;FOLD PLACE 14
;FOLD PROPRIEDADES
MatrizPontos[Pallet_1,Prdt_15CoffeCrisp,14].NumCaixas = 3
MatrizPontos[Pallet_1,Prdt_15CoffeCrisp,14].PickOp = 6
MatrizPontos[Pallet_1,Prdt_15CoffeCrisp,14].ConfGarraOp = 5
MatrizPontos[Pallet_1,Prdt_15CoffeCrisp,14].FechaGarraOp = 0
MatrizPontos[Pallet_1,Prdt_15CoffeCrisp,14].AbreGarraOp = 1
MatrizPontos[Pallet_1,Prdt_15CoffeCrisp,14].SensoresCaixa = 1234
MatrizPontos[Pallet_1,Prdt_15CoffeCrisp,14].TravaGarra = True
MatrizPontos[Pallet_1,Prdt_15CoffeCrisp,14].SkipGoHome = False
MatrizPontos[Pallet_1,Prdt_15CoffeCrisp,14].SkipSobeRelAtual = False
MatrizPontos[Pallet_1,Prdt_15CoffeCrisp,14].XApp1Place=P1_15CoffeCrisp_14_App1
MatrizPontos[Pallet_1,Prdt_15CoffeCrisp,14].XApp2Place=P1_15CoffeCrisp_14_App2
MatrizPontos[Pallet_1,Prdt_15CoffeCrisp,14].XPlace=P1_15CoffeCrisp_14_Place
;ENDFOLD
;FOLD OffsetPlace
MatrizPontos[Pallet_1,Prdt_15CoffeCrisp,14].OffsetPlace.X=0
MatrizPontos[Pallet_1,Prdt_15CoffeCrisp,14].OffsetPlace.Y=0
MatrizPontos[Pallet_1,Prdt_15CoffeCrisp,14].OffsetPlace.Z=0
MatrizPontos[Pallet_1,Prdt_15CoffeCrisp,14].OffsetPlace.A=0
MatrizPontos[Pallet_1,Prdt_15CoffeCrisp,14].OffsetPlace.B=0
MatrizPontos[Pallet_1,Prdt_15CoffeCrisp,14].OffsetPlace.C=0
;ENDFOLD
;ENDFOLD

;ENDFOLD
;ENDFOLD

;FOLD Pallet 1 - Produto 7Aero
;FOLD LAYER 1: PLACE 1 ate 8
;FOLD PLACE 1
;FOLD PROPRIEDADES
MatrizPontos[Pallet_1,Prdt_7Aero,1].NumCaixas = 3
MatrizPontos[Pallet_1,Prdt_7Aero,1].PickOp = 6
MatrizPontos[Pallet_1,Prdt_7Aero,1].ConfGarraOp = 0
MatrizPontos[Pallet_1,Prdt_7Aero,1].FechaGarraOp = 0
MatrizPontos[Pallet_1,Prdt_7Aero,1].AbreGarraOp = 0
MatrizPontos[Pallet_1,Prdt_7Aero,1].SensoresCaixa = 564
MatrizPontos[Pallet_1,Prdt_7Aero,1].TravaGarra = False
MatrizPontos[Pallet_1,Prdt_7Aero,1].SkipGoHome = False
MatrizPontos[Pallet_1,Prdt_7Aero,1].SkipSobeRelAtual = False
MatrizPontos[Pallet_1,Prdt_7Aero,1].XApp1Place=P1_7Aero_1_App1
MatrizPontos[Pallet_1,Prdt_7Aero,1].XApp2Place=P1_7Aero_1_App2
MatrizPontos[Pallet_1,Prdt_7Aero,1].XPlace=P1_7Aero_1_Place
;ENDFOLD
;FOLD OffsetPlace
MatrizPontos[Pallet_1,Prdt_7Aero,1].OffsetPlace.X=0
MatrizPontos[Pallet_1,Prdt_7Aero,1].OffsetPlace.Y=0
MatrizPontos[Pallet_1,Prdt_7Aero,1].OffsetPlace.Z=0
MatrizPontos[Pallet_1,Prdt_7Aero,1].OffsetPlace.A=0
MatrizPontos[Pallet_1,Prdt_7Aero,1].OffsetPlace.B=0
MatrizPontos[Pallet_1,Prdt_7Aero,1].OffsetPlace.C=0
;ENDFOLD
;ENDFOLD

;FOLD PLACE 2
;FOLD PROPRIEDADES
MatrizPontos[Pallet_1,Prdt_7Aero,2].NumCaixas = 3
MatrizPontos[Pallet_1,Prdt_7Aero,2].PickOp = 6
MatrizPontos[Pallet_1,Prdt_7Aero,2].ConfGarraOp = 0
MatrizPontos[Pallet_1,Prdt_7Aero,2].FechaGarraOp = 0
MatrizPontos[Pallet_1,Prdt_7Aero,2].AbreGarraOp = 0
MatrizPontos[Pallet_1,Prdt_7Aero,2].SensoresCaixa = 564
MatrizPontos[Pallet_1,Prdt_7Aero,2].TravaGarra = False
MatrizPontos[Pallet_1,Prdt_7Aero,2].SkipGoHome = False
MatrizPontos[Pallet_1,Prdt_7Aero,2].SkipSobeRelAtual = False
MatrizPontos[Pallet_1,Prdt_7Aero,2].XApp1Place=P1_7Aero_2_App1
MatrizPontos[Pallet_1,Prdt_7Aero,2].XApp2Place=P1_7Aero_2_App2
MatrizPontos[Pallet_1,Prdt_7Aero,2].XPlace=P1_7Aero_2_Place
;ENDFOLD
;FOLD OffsetPlace
MatrizPontos[Pallet_1,Prdt_7Aero,2].OffsetPlace.X=0
MatrizPontos[Pallet_1,Prdt_7Aero,2].OffsetPlace.Y=0
MatrizPontos[Pallet_1,Prdt_7Aero,2].OffsetPlace.Z=0
MatrizPontos[Pallet_1,Prdt_7Aero,2].OffsetPlace.A=0
MatrizPontos[Pallet_1,Prdt_7Aero,2].OffsetPlace.B=0
MatrizPontos[Pallet_1,Prdt_7Aero,2].OffsetPlace.C=0
;ENDFOLD
;ENDFOLD

;FOLD PLACE 3
;FOLD PROPRIEDADES
MatrizPontos[Pallet_1,Prdt_7Aero,3].NumCaixas = 2
MatrizPontos[Pallet_1,Prdt_7Aero,3].PickOp = 8
MatrizPontos[Pallet_1,Prdt_7Aero,3].ConfGarraOp = 5
MatrizPontos[Pallet_1,Prdt_7Aero,3].FechaGarraOp = 0
MatrizPontos[Pallet_1,Prdt_7Aero,3].AbreGarraOp = 0
MatrizPontos[Pallet_1,Prdt_7Aero,3].SensoresCaixa = 12
MatrizPontos[Pallet_1,Prdt_7Aero,3].TravaGarra = False
MatrizPontos[Pallet_1,Prdt_7Aero,3].SkipGoHome = False
MatrizPontos[Pallet_1,Prdt_7Aero,3].SkipSobeRelAtual = False
MatrizPontos[Pallet_1,Prdt_7Aero,3].XApp1Place=P1_7Aero_3_App1
MatrizPontos[Pallet_1,Prdt_7Aero,3].XApp2Place=P1_7Aero_3_App2
MatrizPontos[Pallet_1,Prdt_7Aero,3].XPlace=P1_7Aero_3_Place
;ENDFOLD
;FOLD OffsetPlace
MatrizPontos[Pallet_1,Prdt_7Aero,3].OffsetPlace.X=0
MatrizPontos[Pallet_1,Prdt_7Aero,3].OffsetPlace.Y=0
MatrizPontos[Pallet_1,Prdt_7Aero,3].OffsetPlace.Z=0
MatrizPontos[Pallet_1,Prdt_7Aero,3].OffsetPlace.A=0
MatrizPontos[Pallet_1,Prdt_7Aero,3].OffsetPlace.B=0
MatrizPontos[Pallet_1,Prdt_7Aero,3].OffsetPlace.C=0
;ENDFOLD
;ENDFOLD

;FOLD PLACE 4
;FOLD PROPRIEDADES
MatrizPontos[Pallet_1,Prdt_7Aero,4].NumCaixas = 2
MatrizPontos[Pallet_1,Prdt_7Aero,4].PickOp = 8
MatrizPontos[Pallet_1,Prdt_7Aero,4].ConfGarraOp = 5
MatrizPontos[Pallet_1,Prdt_7Aero,4].FechaGarraOp = 0
MatrizPontos[Pallet_1,Prdt_7Aero,4].AbreGarraOp = 0
MatrizPontos[Pallet_1,Prdt_7Aero,4].SensoresCaixa = 12
MatrizPontos[Pallet_1,Prdt_7Aero,4].TravaGarra = False
MatrizPontos[Pallet_1,Prdt_7Aero,4].SkipGoHome = False
MatrizPontos[Pallet_1,Prdt_7Aero,4].SkipSobeRelAtual = False
MatrizPontos[Pallet_1,Prdt_7Aero,4].XApp1Place=P1_7Aero_4_App1
MatrizPontos[Pallet_1,Prdt_7Aero,4].XApp2Place=P1_7Aero_4_App2
MatrizPontos[Pallet_1,Prdt_7Aero,4].XPlace=P1_7Aero_4_Place
;ENDFOLD
;FOLD OffsetPlace
MatrizPontos[Pallet_1,Prdt_7Aero,4].OffsetPlace.X=0
MatrizPontos[Pallet_1,Prdt_7Aero,4].OffsetPlace.Y=0
MatrizPontos[Pallet_1,Prdt_7Aero,4].OffsetPlace.Z=0
MatrizPontos[Pallet_1,Prdt_7Aero,4].OffsetPlace.A=0
MatrizPontos[Pallet_1,Prdt_7Aero,4].OffsetPlace.B=0
MatrizPontos[Pallet_1,Prdt_7Aero,4].OffsetPlace.C=0
;ENDFOLD
;ENDFOLD

;FOLD PLACE 5
;FOLD PROPRIEDADES
MatrizPontos[Pallet_1,Prdt_7Aero,5].NumCaixas = 3
MatrizPontos[Pallet_1,Prdt_7Aero,5].PickOp = 8
MatrizPontos[Pallet_1,Prdt_7Aero,5].ConfGarraOp = 5
MatrizPontos[Pallet_1,Prdt_7Aero,5].FechaGarraOp = 0
MatrizPontos[Pallet_1,Prdt_7Aero,5].AbreGarraOp = 1
MatrizPontos[Pallet_1,Prdt_7Aero,5].SensoresCaixa = 123
MatrizPontos[Pallet_1,Prdt_7Aero,5].TravaGarra = True
MatrizPontos[Pallet_1,Prdt_7Aero,5].SkipGoHome = False
MatrizPontos[Pallet_1,Prdt_7Aero,5].SkipSobeRelAtual = False
MatrizPontos[Pallet_1,Prdt_7Aero,5].XApp1Place=P1_7Aero_5_App1
MatrizPontos[Pallet_1,Prdt_7Aero,5].XApp2Place=P1_7Aero_5_App2
MatrizPontos[Pallet_1,Prdt_7Aero,5].XPlace=P1_7Aero_5_Place
;ENDFOLD
;FOLD OffsetPlace
MatrizPontos[Pallet_1,Prdt_7Aero,5].OffsetPlace.X=0
MatrizPontos[Pallet_1,Prdt_7Aero,5].OffsetPlace.Y=0
MatrizPontos[Pallet_1,Prdt_7Aero,5].OffsetPlace.Z=0
MatrizPontos[Pallet_1,Prdt_7Aero,5].OffsetPlace.A=0
MatrizPontos[Pallet_1,Prdt_7Aero,5].OffsetPlace.B=0
MatrizPontos[Pallet_1,Prdt_7Aero,5].OffsetPlace.C=0
;ENDFOLD
;ENDFOLD

;FOLD PLACE 6
;FOLD PROPRIEDADES
MatrizPontos[Pallet_1,Prdt_7Aero,6].NumCaixas = 3
MatrizPontos[Pallet_1,Prdt_7Aero,6].PickOp = 8
MatrizPontos[Pallet_1,Prdt_7Aero,6].ConfGarraOp = 5
MatrizPontos[Pallet_1,Prdt_7Aero,6].FechaGarraOp = 0
MatrizPontos[Pallet_1,Prdt_7Aero,6].AbreGarraOp = 1
MatrizPontos[Pallet_1,Prdt_7Aero,6].SensoresCaixa = 123
MatrizPontos[Pallet_1,Prdt_7Aero,6].TravaGarra = True
MatrizPontos[Pallet_1,Prdt_7Aero,6].SkipGoHome = False
MatrizPontos[Pallet_1,Prdt_7Aero,6].SkipSobeRelAtual = False
MatrizPontos[Pallet_1,Prdt_7Aero,6].XApp1Place=P1_7Aero_6_App1
MatrizPontos[Pallet_1,Prdt_7Aero,6].XApp2Place=P1_7Aero_6_App2
MatrizPontos[Pallet_1,Prdt_7Aero,6].XPlace=P1_7Aero_6_Place
;ENDFOLD
;FOLD OffsetPlace
MatrizPontos[Pallet_1,Prdt_7Aero,6].OffsetPlace.X=0
MatrizPontos[Pallet_1,Prdt_7Aero,6].OffsetPlace.Y=0
MatrizPontos[Pallet_1,Prdt_7Aero,6].OffsetPlace.Z=0
MatrizPontos[Pallet_1,Prdt_7Aero,6].OffsetPlace.A=0
MatrizPontos[Pallet_1,Prdt_7Aero,6].OffsetPlace.B=0
MatrizPontos[Pallet_1,Prdt_7Aero,6].OffsetPlace.C=0
;ENDFOLD
;ENDFOLD

;FOLD PLACE 7
;FOLD PROPRIEDADES
MatrizPontos[Pallet_1,Prdt_7Aero,7].NumCaixas = 2
MatrizPontos[Pallet_1,Prdt_7Aero,7].PickOp = 8
MatrizPontos[Pallet_1,Prdt_7Aero,7].ConfGarraOp = 5
MatrizPontos[Pallet_1,Prdt_7Aero,7].FechaGarraOp = 0
MatrizPontos[Pallet_1,Prdt_7Aero,7].AbreGarraOp = 1
MatrizPontos[Pallet_1,Prdt_7Aero,7].SensoresCaixa = 12
MatrizPontos[Pallet_1,Prdt_7Aero,7].TravaGarra = True
MatrizPontos[Pallet_1,Prdt_7Aero,7].SkipGoHome = False
MatrizPontos[Pallet_1,Prdt_7Aero,7].SkipSobeRelAtual = False
MatrizPontos[Pallet_1,Prdt_7Aero,7].XApp1Place=P1_7Aero_7_App1
MatrizPontos[Pallet_1,Prdt_7Aero,7].XApp2Place=P1_7Aero_7_App2
MatrizPontos[Pallet_1,Prdt_7Aero,7].XPlace=P1_7Aero_7_Place
;ENDFOLD
;FOLD OffsetPlace
MatrizPontos[Pallet_1,Prdt_7Aero,7].OffsetPlace.X=0
MatrizPontos[Pallet_1,Prdt_7Aero,7].OffsetPlace.Y=0
MatrizPontos[Pallet_1,Prdt_7Aero,7].OffsetPlace.Z=0
MatrizPontos[Pallet_1,Prdt_7Aero,7].OffsetPlace.A=0
MatrizPontos[Pallet_1,Prdt_7Aero,7].OffsetPlace.B=0
MatrizPontos[Pallet_1,Prdt_7Aero,7].OffsetPlace.C=0
;ENDFOLD
;ENDFOLD

;FOLD PLACE 8
;FOLD PROPRIEDADES
MatrizPontos[Pallet_1,Prdt_7Aero,8].NumCaixas = 2
MatrizPontos[Pallet_1,Prdt_7Aero,8].PickOp = 8
MatrizPontos[Pallet_1,Prdt_7Aero,8].ConfGarraOp = 5
MatrizPontos[Pallet_1,Prdt_7Aero,8].FechaGarraOp = 0
MatrizPontos[Pallet_1,Prdt_7Aero,8].AbreGarraOp = 1
MatrizPontos[Pallet_1,Prdt_7Aero,8].SensoresCaixa = 12
MatrizPontos[Pallet_1,Prdt_7Aero,8].TravaGarra = True
MatrizPontos[Pallet_1,Prdt_7Aero,8].SkipGoHome = False
MatrizPontos[Pallet_1,Prdt_7Aero,8].SkipSobeRelAtual = False
MatrizPontos[Pallet_1,Prdt_7Aero,8].XApp1Place=P1_7Aero_8_App1
MatrizPontos[Pallet_1,Prdt_7Aero,8].XApp2Place=P1_7Aero_8_App2
MatrizPontos[Pallet_1,Prdt_7Aero,8].XPlace=P1_7Aero_8_Place
;ENDFOLD
;FOLD OffsetPlace
MatrizPontos[Pallet_1,Prdt_7Aero,8].OffsetPlace.X=0
MatrizPontos[Pallet_1,Prdt_7Aero,8].OffsetPlace.Y=0
MatrizPontos[Pallet_1,Prdt_7Aero,8].OffsetPlace.Z=0
MatrizPontos[Pallet_1,Prdt_7Aero,8].OffsetPlace.A=0
MatrizPontos[Pallet_1,Prdt_7Aero,8].OffsetPlace.B=0
MatrizPontos[Pallet_1,Prdt_7Aero,8].OffsetPlace.C=0
;ENDFOLD
;ENDFOLD

;ENDFOLD
;FOLD LAYER 2: PLACE 9 ate 16
;FOLD PLACE 9
;FOLD PROPRIEDADES
MatrizPontos[Pallet_1,Prdt_7Aero,9].NumCaixas = 2
MatrizPontos[Pallet_1,Prdt_7Aero,9].PickOp = 8
MatrizPontos[Pallet_1,Prdt_7Aero,9].ConfGarraOp = 5
MatrizPontos[Pallet_1,Prdt_7Aero,9].FechaGarraOp = 0
MatrizPontos[Pallet_1,Prdt_7Aero,9].AbreGarraOp = 1
MatrizPontos[Pallet_1,Prdt_7Aero,9].SensoresCaixa = 12
MatrizPontos[Pallet_1,Prdt_7Aero,9].TravaGarra = True
MatrizPontos[Pallet_1,Prdt_7Aero,9].SkipGoHome = False
MatrizPontos[Pallet_1,Prdt_7Aero,9].SkipSobeRelAtual = False
MatrizPontos[Pallet_1,Prdt_7Aero,9].XApp1Place=P1_7Aero_9_App1
MatrizPontos[Pallet_1,Prdt_7Aero,9].XApp2Place=P1_7Aero_9_App2
MatrizPontos[Pallet_1,Prdt_7Aero,9].XPlace=P1_7Aero_9_Place
;ENDFOLD
;FOLD OffsetPlace
MatrizPontos[Pallet_1,Prdt_7Aero,9].OffsetPlace.X=0
MatrizPontos[Pallet_1,Prdt_7Aero,9].OffsetPlace.Y=0
MatrizPontos[Pallet_1,Prdt_7Aero,9].OffsetPlace.Z=0
MatrizPontos[Pallet_1,Prdt_7Aero,9].OffsetPlace.A=0
MatrizPontos[Pallet_1,Prdt_7Aero,9].OffsetPlace.B=0
MatrizPontos[Pallet_1,Prdt_7Aero,9].OffsetPlace.C=0
;ENDFOLD
;ENDFOLD

;FOLD PLACE 10
;FOLD PROPRIEDADES
MatrizPontos[Pallet_1,Prdt_7Aero,10].NumCaixas = 2
MatrizPontos[Pallet_1,Prdt_7Aero,10].PickOp = 8
MatrizPontos[Pallet_1,Prdt_7Aero,10].ConfGarraOp = 5
MatrizPontos[Pallet_1,Prdt_7Aero,10].FechaGarraOp = 0
MatrizPontos[Pallet_1,Prdt_7Aero,10].AbreGarraOp = 1
MatrizPontos[Pallet_1,Prdt_7Aero,10].SensoresCaixa = 12
MatrizPontos[Pallet_1,Prdt_7Aero,10].TravaGarra = True
MatrizPontos[Pallet_1,Prdt_7Aero,10].SkipGoHome = False
MatrizPontos[Pallet_1,Prdt_7Aero,10].SkipSobeRelAtual = False
MatrizPontos[Pallet_1,Prdt_7Aero,10].XApp1Place=P1_7Aero_10_App1
MatrizPontos[Pallet_1,Prdt_7Aero,10].XApp2Place=P1_7Aero_10_App2
MatrizPontos[Pallet_1,Prdt_7Aero,10].XPlace=P1_7Aero_10_Place
;ENDFOLD
;FOLD OffsetPlace
MatrizPontos[Pallet_1,Prdt_7Aero,10].OffsetPlace.X=0
MatrizPontos[Pallet_1,Prdt_7Aero,10].OffsetPlace.Y=0
MatrizPontos[Pallet_1,Prdt_7Aero,10].OffsetPlace.Z=0
MatrizPontos[Pallet_1,Prdt_7Aero,10].OffsetPlace.A=0
MatrizPontos[Pallet_1,Prdt_7Aero,10].OffsetPlace.B=0
MatrizPontos[Pallet_1,Prdt_7Aero,10].OffsetPlace.C=0
;ENDFOLD
;ENDFOLD

;FOLD PLACE 11
;FOLD PROPRIEDADES
MatrizPontos[Pallet_1,Prdt_7Aero,11].NumCaixas = 3
MatrizPontos[Pallet_1,Prdt_7Aero,11].PickOp = 8
MatrizPontos[Pallet_1,Prdt_7Aero,11].ConfGarraOp = 5
MatrizPontos[Pallet_1,Prdt_7Aero,11].FechaGarraOp = 0
MatrizPontos[Pallet_1,Prdt_7Aero,11].AbreGarraOp = 0
MatrizPontos[Pallet_1,Prdt_7Aero,11].SensoresCaixa = 123
MatrizPontos[Pallet_1,Prdt_7Aero,11].TravaGarra = False
MatrizPontos[Pallet_1,Prdt_7Aero,11].SkipGoHome = False
MatrizPontos[Pallet_1,Prdt_7Aero,11].SkipSobeRelAtual = False
MatrizPontos[Pallet_1,Prdt_7Aero,11].XApp1Place=P1_7Aero_11_App1
MatrizPontos[Pallet_1,Prdt_7Aero,11].XApp2Place=P1_7Aero_11_App2
MatrizPontos[Pallet_1,Prdt_7Aero,11].XPlace=P1_7Aero_11_Place
;ENDFOLD
;FOLD OffsetPlace
MatrizPontos[Pallet_1,Prdt_7Aero,11].OffsetPlace.X=0
MatrizPontos[Pallet_1,Prdt_7Aero,11].OffsetPlace.Y=0
MatrizPontos[Pallet_1,Prdt_7Aero,11].OffsetPlace.Z=0
MatrizPontos[Pallet_1,Prdt_7Aero,11].OffsetPlace.A=0
MatrizPontos[Pallet_1,Prdt_7Aero,11].OffsetPlace.B=0
MatrizPontos[Pallet_1,Prdt_7Aero,11].OffsetPlace.C=0
;ENDFOLD
;ENDFOLD

;FOLD PLACE 12
;FOLD PROPRIEDADES
MatrizPontos[Pallet_1,Prdt_7Aero,12].NumCaixas = 3
MatrizPontos[Pallet_1,Prdt_7Aero,12].PickOp = 8
MatrizPontos[Pallet_1,Prdt_7Aero,12].ConfGarraOp = 5
MatrizPontos[Pallet_1,Prdt_7Aero,12].FechaGarraOp = 0
MatrizPontos[Pallet_1,Prdt_7Aero,12].AbreGarraOp = 0
MatrizPontos[Pallet_1,Prdt_7Aero,12].SensoresCaixa = 123
MatrizPontos[Pallet_1,Prdt_7Aero,12].TravaGarra = False
MatrizPontos[Pallet_1,Prdt_7Aero,12].SkipGoHome = False
MatrizPontos[Pallet_1,Prdt_7Aero,12].SkipSobeRelAtual = False
MatrizPontos[Pallet_1,Prdt_7Aero,12].XApp1Place=P1_7Aero_12_App1
MatrizPontos[Pallet_1,Prdt_7Aero,12].XApp2Place=P1_7Aero_12_App2
MatrizPontos[Pallet_1,Prdt_7Aero,12].XPlace=P1_7Aero_12_Place
;ENDFOLD
;FOLD OffsetPlace
MatrizPontos[Pallet_1,Prdt_7Aero,12].OffsetPlace.X=0
MatrizPontos[Pallet_1,Prdt_7Aero,12].OffsetPlace.Y=0
MatrizPontos[Pallet_1,Prdt_7Aero,12].OffsetPlace.Z=0
MatrizPontos[Pallet_1,Prdt_7Aero,12].OffsetPlace.A=0
MatrizPontos[Pallet_1,Prdt_7Aero,12].OffsetPlace.B=0
MatrizPontos[Pallet_1,Prdt_7Aero,12].OffsetPlace.C=0
;ENDFOLD
;ENDFOLD

;FOLD PLACE 13
;FOLD PROPRIEDADES
MatrizPontos[Pallet_1,Prdt_7Aero,13].NumCaixas = 3
MatrizPontos[Pallet_1,Prdt_7Aero,13].PickOp = 8
MatrizPontos[Pallet_1,Prdt_7Aero,13].ConfGarraOp = 5
MatrizPontos[Pallet_1,Prdt_7Aero,13].FechaGarraOp = 0
MatrizPontos[Pallet_1,Prdt_7Aero,13].AbreGarraOp = 0
MatrizPontos[Pallet_1,Prdt_7Aero,13].SensoresCaixa = 123
MatrizPontos[Pallet_1,Prdt_7Aero,13].TravaGarra = False
MatrizPontos[Pallet_1,Prdt_7Aero,13].SkipGoHome = False
MatrizPontos[Pallet_1,Prdt_7Aero,13].SkipSobeRelAtual = False
MatrizPontos[Pallet_1,Prdt_7Aero,13].XApp1Place=P1_7Aero_13_App1
MatrizPontos[Pallet_1,Prdt_7Aero,13].XApp2Place=P1_7Aero_13_App2
MatrizPontos[Pallet_1,Prdt_7Aero,13].XPlace=P1_7Aero_13_Place
;ENDFOLD
;FOLD OffsetPlace
MatrizPontos[Pallet_1,Prdt_7Aero,13].OffsetPlace.X=0
MatrizPontos[Pallet_1,Prdt_7Aero,13].OffsetPlace.Y=0
MatrizPontos[Pallet_1,Prdt_7Aero,13].OffsetPlace.Z=0
MatrizPontos[Pallet_1,Prdt_7Aero,13].OffsetPlace.A=0
MatrizPontos[Pallet_1,Prdt_7Aero,13].OffsetPlace.B=0
MatrizPontos[Pallet_1,Prdt_7Aero,13].OffsetPlace.C=0
;ENDFOLD
;ENDFOLD

;FOLD PLACE 14
;FOLD PROPRIEDADES
MatrizPontos[Pallet_1,Prdt_7Aero,14].NumCaixas = 3
MatrizPontos[Pallet_1,Prdt_7Aero,14].PickOp = 8
MatrizPontos[Pallet_1,Prdt_7Aero,14].ConfGarraOp = 5
MatrizPontos[Pallet_1,Prdt_7Aero,14].FechaGarraOp = 0
MatrizPontos[Pallet_1,Prdt_7Aero,14].AbreGarraOp = 0
MatrizPontos[Pallet_1,Prdt_7Aero,14].SensoresCaixa = 123
MatrizPontos[Pallet_1,Prdt_7Aero,14].TravaGarra = False
MatrizPontos[Pallet_1,Prdt_7Aero,14].SkipGoHome = False
MatrizPontos[Pallet_1,Prdt_7Aero,14].SkipSobeRelAtual = False
MatrizPontos[Pallet_1,Prdt_7Aero,14].XApp1Place=P1_7Aero_14_App1
MatrizPontos[Pallet_1,Prdt_7Aero,14].XApp2Place=P1_7Aero_14_App2
MatrizPontos[Pallet_1,Prdt_7Aero,14].XPlace=P1_7Aero_14_Place
;ENDFOLD
;FOLD OffsetPlace
MatrizPontos[Pallet_1,Prdt_7Aero,14].OffsetPlace.X=0
MatrizPontos[Pallet_1,Prdt_7Aero,14].OffsetPlace.Y=0
MatrizPontos[Pallet_1,Prdt_7Aero,14].OffsetPlace.Z=0
MatrizPontos[Pallet_1,Prdt_7Aero,14].OffsetPlace.A=0
MatrizPontos[Pallet_1,Prdt_7Aero,14].OffsetPlace.B=0
MatrizPontos[Pallet_1,Prdt_7Aero,14].OffsetPlace.C=0
;ENDFOLD
;ENDFOLD

;FOLD PLACE 15
;FOLD PROPRIEDADES
MatrizPontos[Pallet_1,Prdt_7Aero,15].NumCaixas = 2
MatrizPontos[Pallet_1,Prdt_7Aero,15].PickOp = 8
MatrizPontos[Pallet_1,Prdt_7Aero,15].ConfGarraOp = 5
MatrizPontos[Pallet_1,Prdt_7Aero,15].FechaGarraOp = 0
MatrizPontos[Pallet_1,Prdt_7Aero,15].AbreGarraOp = 1
MatrizPontos[Pallet_1,Prdt_7Aero,15].SensoresCaixa = 12
MatrizPontos[Pallet_1,Prdt_7Aero,15].TravaGarra = True
MatrizPontos[Pallet_1,Prdt_7Aero,15].SkipGoHome = False
MatrizPontos[Pallet_1,Prdt_7Aero,15].SkipSobeRelAtual = False
MatrizPontos[Pallet_1,Prdt_7Aero,15].XApp1Place=P1_7Aero_15_App1
MatrizPontos[Pallet_1,Prdt_7Aero,15].XApp2Place=P1_7Aero_15_App2
MatrizPontos[Pallet_1,Prdt_7Aero,15].XPlace=P1_7Aero_15_Place
;ENDFOLD
;FOLD OffsetPlace
MatrizPontos[Pallet_1,Prdt_7Aero,15].OffsetPlace.X=0
MatrizPontos[Pallet_1,Prdt_7Aero,15].OffsetPlace.Y=0
MatrizPontos[Pallet_1,Prdt_7Aero,15].OffsetPlace.Z=0
MatrizPontos[Pallet_1,Prdt_7Aero,15].OffsetPlace.A=0
MatrizPontos[Pallet_1,Prdt_7Aero,15].OffsetPlace.B=0
MatrizPontos[Pallet_1,Prdt_7Aero,15].OffsetPlace.C=0
;ENDFOLD
;ENDFOLD

;FOLD PLACE 16
;FOLD PROPRIEDADES
MatrizPontos[Pallet_1,Prdt_7Aero,16].NumCaixas = 2
MatrizPontos[Pallet_1,Prdt_7Aero,16].PickOp = 8
MatrizPontos[Pallet_1,Prdt_7Aero,16].ConfGarraOp = 5
MatrizPontos[Pallet_1,Prdt_7Aero,16].FechaGarraOp = 0
MatrizPontos[Pallet_1,Prdt_7Aero,16].AbreGarraOp = 1
MatrizPontos[Pallet_1,Prdt_7Aero,16].SensoresCaixa = 12
MatrizPontos[Pallet_1,Prdt_7Aero,16].TravaGarra = True
MatrizPontos[Pallet_1,Prdt_7Aero,16].SkipGoHome = False
MatrizPontos[Pallet_1,Prdt_7Aero,16].SkipSobeRelAtual = False
MatrizPontos[Pallet_1,Prdt_7Aero,16].XApp1Place=P1_7Aero_16_App1
MatrizPontos[Pallet_1,Prdt_7Aero,16].XApp2Place=P1_7Aero_16_App2
MatrizPontos[Pallet_1,Prdt_7Aero,16].XPlace=P1_7Aero_16_Place
;ENDFOLD
;FOLD OffsetPlace
MatrizPontos[Pallet_1,Prdt_7Aero,16].OffsetPlace.X=0
MatrizPontos[Pallet_1,Prdt_7Aero,16].OffsetPlace.Y=0
MatrizPontos[Pallet_1,Prdt_7Aero,16].OffsetPlace.Z=0
MatrizPontos[Pallet_1,Prdt_7Aero,16].OffsetPlace.A=0
MatrizPontos[Pallet_1,Prdt_7Aero,16].OffsetPlace.B=0
MatrizPontos[Pallet_1,Prdt_7Aero,16].OffsetPlace.C=0
;ENDFOLD
;ENDFOLD

;ENDFOLD
;ENDFOLD

;FOLD Pallet 1 - Produto 32BarPacking
;FOLD LAYER 1: PLACE 1 ate 3
;FOLD PLACE 1
;FOLD PROPRIEDADES
MatrizPontos[Pallet_1,Prdt_32BarPacking,1].NumCaixas = 3
MatrizPontos[Pallet_1,Prdt_32BarPacking,1].PickOp = 2
MatrizPontos[Pallet_1,Prdt_32BarPacking,1].ConfGarraOp = 3
MatrizPontos[Pallet_1,Prdt_32BarPacking,1].FechaGarraOp = 0
MatrizPontos[Pallet_1,Prdt_32BarPacking,1].AbreGarraOp = 0
MatrizPontos[Pallet_1,Prdt_32BarPacking,1].SensoresCaixa = 12345
MatrizPontos[Pallet_1,Prdt_32BarPacking,1].TravaGarra = False
MatrizPontos[Pallet_1,Prdt_32BarPacking,1].SkipGoHome = False
MatrizPontos[Pallet_1,Prdt_32BarPacking,1].SkipSobeRelAtual = False
MatrizPontos[Pallet_1,Prdt_32BarPacking,1].XApp1Place=P1_32BarPacking_1_App1
MatrizPontos[Pallet_1,Prdt_32BarPacking,1].XApp2Place=P1_32BarPacking_1_App2
MatrizPontos[Pallet_1,Prdt_32BarPacking,1].XPlace=P1_32BarPacking_1_Place
;ENDFOLD
;FOLD OffsetPlace
MatrizPontos[Pallet_1,Prdt_32BarPacking,1].OffsetPlace.X=0
MatrizPontos[Pallet_1,Prdt_32BarPacking,1].OffsetPlace.Y=0
MatrizPontos[Pallet_1,Prdt_32BarPacking,1].OffsetPlace.Z=0
MatrizPontos[Pallet_1,Prdt_32BarPacking,1].OffsetPlace.A=0
MatrizPontos[Pallet_1,Prdt_32BarPacking,1].OffsetPlace.B=0
MatrizPontos[Pallet_1,Prdt_32BarPacking,1].OffsetPlace.C=0
;ENDFOLD
;ENDFOLD

;FOLD PLACE 2
;FOLD PROPRIEDADES
MatrizPontos[Pallet_1,Prdt_32BarPacking,2].NumCaixas = 3
MatrizPontos[Pallet_1,Prdt_32BarPacking,2].PickOp = 2
MatrizPontos[Pallet_1,Prdt_32BarPacking,2].ConfGarraOp = 3
MatrizPontos[Pallet_1,Prdt_32BarPacking,2].FechaGarraOp = 0
MatrizPontos[Pallet_1,Prdt_32BarPacking,2].AbreGarraOp = 0
MatrizPontos[Pallet_1,Prdt_32BarPacking,2].SensoresCaixa = 12345
MatrizPontos[Pallet_1,Prdt_32BarPacking,2].TravaGarra = False
MatrizPontos[Pallet_1,Prdt_32BarPacking,2].SkipGoHome = False
MatrizPontos[Pallet_1,Prdt_32BarPacking,2].SkipSobeRelAtual = False
MatrizPontos[Pallet_1,Prdt_32BarPacking,2].XApp1Place=P1_32BarPacking_2_App1
MatrizPontos[Pallet_1,Prdt_32BarPacking,2].XApp2Place=P1_32BarPacking_2_App2
MatrizPontos[Pallet_1,Prdt_32BarPacking,2].XPlace=P1_32BarPacking_2_Place
;ENDFOLD
;FOLD OffsetPlace
MatrizPontos[Pallet_1,Prdt_32BarPacking,2].OffsetPlace.X=0
MatrizPontos[Pallet_1,Prdt_32BarPacking,2].OffsetPlace.Y=0
MatrizPontos[Pallet_1,Prdt_32BarPacking,2].OffsetPlace.Z=0
MatrizPontos[Pallet_1,Prdt_32BarPacking,2].OffsetPlace.A=0
MatrizPontos[Pallet_1,Prdt_32BarPacking,2].OffsetPlace.B=0
MatrizPontos[Pallet_1,Prdt_32BarPacking,2].OffsetPlace.C=0
;ENDFOLD
;ENDFOLD

;FOLD PLACE 3
;FOLD PROPRIEDADES
MatrizPontos[Pallet_1,Prdt_32BarPacking,3].NumCaixas = 3
MatrizPontos[Pallet_1,Prdt_32BarPacking,3].PickOp = 2
MatrizPontos[Pallet_1,Prdt_32BarPacking,3].ConfGarraOp = 3
MatrizPontos[Pallet_1,Prdt_32BarPacking,3].FechaGarraOp = 0
MatrizPontos[Pallet_1,Prdt_32BarPacking,3].AbreGarraOp = 0
MatrizPontos[Pallet_1,Prdt_32BarPacking,3].SensoresCaixa = 12345
MatrizPontos[Pallet_1,Prdt_32BarPacking,3].TravaGarra = False
MatrizPontos[Pallet_1,Prdt_32BarPacking,3].SkipGoHome = False
MatrizPontos[Pallet_1,Prdt_32BarPacking,3].SkipSobeRelAtual = False
MatrizPontos[Pallet_1,Prdt_32BarPacking,3].XApp1Place=P1_32BarPacking_3_App1
MatrizPontos[Pallet_1,Prdt_32BarPacking,3].XApp2Place=P1_32BarPacking_3_App2
MatrizPontos[Pallet_1,Prdt_32BarPacking,3].XPlace=P1_32BarPacking_3_Place
;ENDFOLD
;FOLD OffsetPlace
MatrizPontos[Pallet_1,Prdt_32BarPacking,3].OffsetPlace.X=0
MatrizPontos[Pallet_1,Prdt_32BarPacking,3].OffsetPlace.Y=0
MatrizPontos[Pallet_1,Prdt_32BarPacking,3].OffsetPlace.Z=0
MatrizPontos[Pallet_1,Prdt_32BarPacking,3].OffsetPlace.A=0
MatrizPontos[Pallet_1,Prdt_32BarPacking,3].OffsetPlace.B=0
MatrizPontos[Pallet_1,Prdt_32BarPacking,3].OffsetPlace.C=0
;ENDFOLD
;ENDFOLD

;ENDFOLD
;ENDFOLD

;FOLD Pallet 1 - Produto 33BarPacking
;FOLD LAYER 1: PLACE 1 ate 2
;FOLD PLACE 1
;FOLD PROPRIEDADES
MatrizPontos[Pallet_1,Prdt_33BarPacking,1].NumCaixas = 3
MatrizPontos[Pallet_1,Prdt_33BarPacking,1].PickOp = 2
MatrizPontos[Pallet_1,Prdt_33BarPacking,1].ConfGarraOp = 2
MatrizPontos[Pallet_1,Prdt_33BarPacking,1].FechaGarraOp = 0
MatrizPontos[Pallet_1,Prdt_33BarPacking,1].AbreGarraOp = 0
MatrizPontos[Pallet_1,Prdt_33BarPacking,1].SensoresCaixa = 12345
MatrizPontos[Pallet_1,Prdt_33BarPacking,1].TravaGarra = False
MatrizPontos[Pallet_1,Prdt_33BarPacking,1].SkipGoHome = False
MatrizPontos[Pallet_1,Prdt_33BarPacking,1].SkipSobeRelAtual = False
MatrizPontos[Pallet_1,Prdt_33BarPacking,1].XApp1Place=P1_33BarPacking_1_App1
MatrizPontos[Pallet_1,Prdt_33BarPacking,1].XApp2Place=P1_33BarPacking_1_App2
MatrizPontos[Pallet_1,Prdt_33BarPacking,1].XPlace=P1_33BarPacking_1_Place
;ENDFOLD
;FOLD OffsetPlace
MatrizPontos[Pallet_1,Prdt_33BarPacking,1].OffsetPlace.X=0
MatrizPontos[Pallet_1,Prdt_33BarPacking,1].OffsetPlace.Y=0
MatrizPontos[Pallet_1,Prdt_33BarPacking,1].OffsetPlace.Z=0
MatrizPontos[Pallet_1,Prdt_33BarPacking,1].OffsetPlace.A=0
MatrizPontos[Pallet_1,Prdt_33BarPacking,1].OffsetPlace.B=0
MatrizPontos[Pallet_1,Prdt_33BarPacking,1].OffsetPlace.C=0
;ENDFOLD
;ENDFOLD

;FOLD PLACE 2
;FOLD PROPRIEDADES
MatrizPontos[Pallet_1,Prdt_33BarPacking,2].NumCaixas = 3
MatrizPontos[Pallet_1,Prdt_33BarPacking,2].PickOp = 2
MatrizPontos[Pallet_1,Prdt_33BarPacking,2].ConfGarraOp = 2
MatrizPontos[Pallet_1,Prdt_33BarPacking,2].FechaGarraOp = 0
MatrizPontos[Pallet_1,Prdt_33BarPacking,2].AbreGarraOp = 0
MatrizPontos[Pallet_1,Prdt_33BarPacking,2].SensoresCaixa = 12345
MatrizPontos[Pallet_1,Prdt_33BarPacking,2].TravaGarra = False
MatrizPontos[Pallet_1,Prdt_33BarPacking,2].SkipGoHome = False
MatrizPontos[Pallet_1,Prdt_33BarPacking,2].SkipSobeRelAtual = False
MatrizPontos[Pallet_1,Prdt_33BarPacking,2].XApp1Place=P1_33BarPacking_2_App1
MatrizPontos[Pallet_1,Prdt_33BarPacking,2].XApp2Place=P1_33BarPacking_2_App2
MatrizPontos[Pallet_1,Prdt_33BarPacking,2].XPlace=P1_33BarPacking_2_Place
;ENDFOLD
;FOLD OffsetPlace
MatrizPontos[Pallet_1,Prdt_33BarPacking,2].OffsetPlace.X=0
MatrizPontos[Pallet_1,Prdt_33BarPacking,2].OffsetPlace.Y=0
MatrizPontos[Pallet_1,Prdt_33BarPacking,2].OffsetPlace.Z=0
MatrizPontos[Pallet_1,Prdt_33BarPacking,2].OffsetPlace.A=0
MatrizPontos[Pallet_1,Prdt_33BarPacking,2].OffsetPlace.B=0
MatrizPontos[Pallet_1,Prdt_33BarPacking,2].OffsetPlace.C=0
;ENDFOLD
;ENDFOLD

;ENDFOLD
;ENDFOLD

;FOLD Pallet 1 - Produto 37BarPacking
;FOLD LAYER 1: PLACE 1 ate 2
;FOLD PLACE 1
;FOLD PROPRIEDADES
MatrizPontos[Pallet_1,Prdt_37BarPacking,1].NumCaixas = 3
MatrizPontos[Pallet_1,Prdt_37BarPacking,1].PickOp = 2
MatrizPontos[Pallet_1,Prdt_37BarPacking,1].ConfGarraOp = 2
MatrizPontos[Pallet_1,Prdt_37BarPacking,1].FechaGarraOp = 0
MatrizPontos[Pallet_1,Prdt_37BarPacking,1].AbreGarraOp = 0
MatrizPontos[Pallet_1,Prdt_37BarPacking,1].SensoresCaixa = 123456
MatrizPontos[Pallet_1,Prdt_37BarPacking,1].TravaGarra = False
MatrizPontos[Pallet_1,Prdt_37BarPacking,1].SkipGoHome = False
MatrizPontos[Pallet_1,Prdt_37BarPacking,1].SkipSobeRelAtual = False
MatrizPontos[Pallet_1,Prdt_37BarPacking,1].XApp1Place=P1_37BarPacking_1_App1
MatrizPontos[Pallet_1,Prdt_37BarPacking,1].XApp2Place=P1_37BarPacking_1_App2
MatrizPontos[Pallet_1,Prdt_37BarPacking,1].XPlace=P1_37BarPacking_1_Place
;ENDFOLD
;FOLD OffsetPlace
MatrizPontos[Pallet_1,Prdt_37BarPacking,1].OffsetPlace.X=0
MatrizPontos[Pallet_1,Prdt_37BarPacking,1].OffsetPlace.Y=0
MatrizPontos[Pallet_1,Prdt_37BarPacking,1].OffsetPlace.Z=0
MatrizPontos[Pallet_1,Prdt_37BarPacking,1].OffsetPlace.A=0
MatrizPontos[Pallet_1,Prdt_37BarPacking,1].OffsetPlace.B=0
MatrizPontos[Pallet_1,Prdt_37BarPacking,1].OffsetPlace.C=0
;ENDFOLD
;ENDFOLD

;FOLD PLACE 2
;FOLD PROPRIEDADES
MatrizPontos[Pallet_1,Prdt_37BarPacking,2].NumCaixas = 3
MatrizPontos[Pallet_1,Prdt_37BarPacking,2].PickOp = 2
MatrizPontos[Pallet_1,Prdt_37BarPacking,2].ConfGarraOp = 2
MatrizPontos[Pallet_1,Prdt_37BarPacking,2].FechaGarraOp = 0
MatrizPontos[Pallet_1,Prdt_37BarPacking,2].AbreGarraOp = 0
MatrizPontos[Pallet_1,Prdt_37BarPacking,2].SensoresCaixa = 123456
MatrizPontos[Pallet_1,Prdt_37BarPacking,2].TravaGarra = False
MatrizPontos[Pallet_1,Prdt_37BarPacking,2].SkipGoHome = False
MatrizPontos[Pallet_1,Prdt_37BarPacking,2].SkipSobeRelAtual = False
MatrizPontos[Pallet_1,Prdt_37BarPacking,2].XApp1Place=P1_37BarPacking_2_App1
MatrizPontos[Pallet_1,Prdt_37BarPacking,2].XApp2Place=P1_37BarPacking_2_App2
MatrizPontos[Pallet_1,Prdt_37BarPacking,2].XPlace=P1_37BarPacking_2_Place
;ENDFOLD
;FOLD OffsetPlace
MatrizPontos[Pallet_1,Prdt_37BarPacking,2].OffsetPlace.X=0
MatrizPontos[Pallet_1,Prdt_37BarPacking,2].OffsetPlace.Y=0
MatrizPontos[Pallet_1,Prdt_37BarPacking,2].OffsetPlace.Z=0
MatrizPontos[Pallet_1,Prdt_37BarPacking,2].OffsetPlace.A=0
MatrizPontos[Pallet_1,Prdt_37BarPacking,2].OffsetPlace.B=0
MatrizPontos[Pallet_1,Prdt_37BarPacking,2].OffsetPlace.C=0
;ENDFOLD
;ENDFOLD

;ENDFOLD
;ENDFOLD

;FOLD Pallet 1 - Produto 36BarPacking
;FOLD LAYER 1: PLACE 1 ate 1
;FOLD PLACE 1
;FOLD PROPRIEDADES
MatrizPontos[Pallet_1,Prdt_36BarPacking,1].NumCaixas = 3
MatrizPontos[Pallet_1,Prdt_36BarPacking,1].PickOp = 2
MatrizPontos[Pallet_1,Prdt_36BarPacking,1].ConfGarraOp = 2
MatrizPontos[Pallet_1,Prdt_36BarPacking,1].FechaGarraOp = 0
MatrizPontos[Pallet_1,Prdt_36BarPacking,1].AbreGarraOp = 0
MatrizPontos[Pallet_1,Prdt_36BarPacking,1].SensoresCaixa = 123456
MatrizPontos[Pallet_1,Prdt_36BarPacking,1].TravaGarra = False
MatrizPontos[Pallet_1,Prdt_36BarPacking,1].SkipGoHome = False
MatrizPontos[Pallet_1,Prdt_36BarPacking,1].SkipSobeRelAtual = False
MatrizPontos[Pallet_1,Prdt_36BarPacking,1].XApp1Place=P1_36BarPacking_1_App1
MatrizPontos[Pallet_1,Prdt_36BarPacking,1].XApp2Place=P1_36BarPacking_1_App2
MatrizPontos[Pallet_1,Prdt_36BarPacking,1].XPlace=P1_36BarPacking_1_Place
;ENDFOLD
;FOLD OffsetPlace
MatrizPontos[Pallet_1,Prdt_36BarPacking,1].OffsetPlace.X=0
MatrizPontos[Pallet_1,Prdt_36BarPacking,1].OffsetPlace.Y=0
MatrizPontos[Pallet_1,Prdt_36BarPacking,1].OffsetPlace.Z=0
MatrizPontos[Pallet_1,Prdt_36BarPacking,1].OffsetPlace.A=0
MatrizPontos[Pallet_1,Prdt_36BarPacking,1].OffsetPlace.B=0
MatrizPontos[Pallet_1,Prdt_36BarPacking,1].OffsetPlace.C=0
;ENDFOLD
;ENDFOLD

;ENDFOLD
;ENDFOLD

;FOLD Pallet 1 - Produto 34BarPacking
;FOLD LAYER 1: PLACE 1 ate 2
;FOLD PLACE 1
;FOLD PROPRIEDADES
MatrizPontos[Pallet_1,Prdt_34BarPacking,1].NumCaixas = 1
MatrizPontos[Pallet_1,Prdt_34BarPacking,1].PickOp = 3
MatrizPontos[Pallet_1,Prdt_34BarPacking,1].ConfGarraOp = 3
MatrizPontos[Pallet_1,Prdt_34BarPacking,1].FechaGarraOp = 0
MatrizPontos[Pallet_1,Prdt_34BarPacking,1].AbreGarraOp = 0
MatrizPontos[Pallet_1,Prdt_34BarPacking,1].SensoresCaixa = 123
MatrizPontos[Pallet_1,Prdt_34BarPacking,1].TravaGarra = False
MatrizPontos[Pallet_1,Prdt_34BarPacking,1].SkipGoHome = False
MatrizPontos[Pallet_1,Prdt_34BarPacking,1].SkipSobeRelAtual = False
MatrizPontos[Pallet_1,Prdt_34BarPacking,1].XApp1Place=P1_34BarPacking_1_App1
MatrizPontos[Pallet_1,Prdt_34BarPacking,1].XApp2Place=P1_34BarPacking_1_App2
MatrizPontos[Pallet_1,Prdt_34BarPacking,1].XPlace=P1_34BarPacking_1_Place
;ENDFOLD
;FOLD OffsetPlace
MatrizPontos[Pallet_1,Prdt_34BarPacking,1].OffsetPlace.X=0
MatrizPontos[Pallet_1,Prdt_34BarPacking,1].OffsetPlace.Y=0
MatrizPontos[Pallet_1,Prdt_34BarPacking,1].OffsetPlace.Z=0
MatrizPontos[Pallet_1,Prdt_34BarPacking,1].OffsetPlace.A=0
MatrizPontos[Pallet_1,Prdt_34BarPacking,1].OffsetPlace.B=0
MatrizPontos[Pallet_1,Prdt_34BarPacking,1].OffsetPlace.C=0
;ENDFOLD
;ENDFOLD

;FOLD PLACE 2
;FOLD PROPRIEDADES
MatrizPontos[Pallet_1,Prdt_34BarPacking,2].NumCaixas = 1
MatrizPontos[Pallet_1,Prdt_34BarPacking,2].PickOp = 3
MatrizPontos[Pallet_1,Prdt_34BarPacking,2].ConfGarraOp = 3
MatrizPontos[Pallet_1,Prdt_34BarPacking,2].FechaGarraOp = 0
MatrizPontos[Pallet_1,Prdt_34BarPacking,2].AbreGarraOp = 0
MatrizPontos[Pallet_1,Prdt_34BarPacking,2].SensoresCaixa = 123
MatrizPontos[Pallet_1,Prdt_34BarPacking,2].TravaGarra = False
MatrizPontos[Pallet_1,Prdt_34BarPacking,2].SkipGoHome = False
MatrizPontos[Pallet_1,Prdt_34BarPacking,2].SkipSobeRelAtual = False
MatrizPontos[Pallet_1,Prdt_34BarPacking,2].XApp1Place=P1_34BarPacking_2_App1
MatrizPontos[Pallet_1,Prdt_34BarPacking,2].XApp2Place=P1_34BarPacking_2_App2
MatrizPontos[Pallet_1,Prdt_34BarPacking,2].XPlace=P1_34BarPacking_2_Place
;ENDFOLD
;FOLD OffsetPlace
MatrizPontos[Pallet_1,Prdt_34BarPacking,2].OffsetPlace.X=0
MatrizPontos[Pallet_1,Prdt_34BarPacking,2].OffsetPlace.Y=0
MatrizPontos[Pallet_1,Prdt_34BarPacking,2].OffsetPlace.Z=0
MatrizPontos[Pallet_1,Prdt_34BarPacking,2].OffsetPlace.A=0
MatrizPontos[Pallet_1,Prdt_34BarPacking,2].OffsetPlace.B=0
MatrizPontos[Pallet_1,Prdt_34BarPacking,2].OffsetPlace.C=0
;ENDFOLD
;ENDFOLD

;ENDFOLD
;ENDFOLD

;FOLD Pallet 1 - Produto 35BarPacking
;FOLD LAYER 1: PLACE 1 ate 3
;FOLD PLACE 1
;FOLD PROPRIEDADES
MatrizPontos[Pallet_1,Prdt_35BarPacking,1].NumCaixas = 1
MatrizPontos[Pallet_1,Prdt_35BarPacking,1].PickOp = 2
MatrizPontos[Pallet_1,Prdt_35BarPacking,1].ConfGarraOp = 2
MatrizPontos[Pallet_1,Prdt_35BarPacking,1].FechaGarraOp = 0
MatrizPontos[Pallet_1,Prdt_35BarPacking,1].AbreGarraOp = 0
MatrizPontos[Pallet_1,Prdt_35BarPacking,1].SensoresCaixa = 12
MatrizPontos[Pallet_1,Prdt_35BarPacking,1].TravaGarra = False
MatrizPontos[Pallet_1,Prdt_35BarPacking,1].SkipGoHome = False
MatrizPontos[Pallet_1,Prdt_35BarPacking,1].SkipSobeRelAtual = False
MatrizPontos[Pallet_1,Prdt_35BarPacking,1].XApp1Place=P1_35BarPacking_1_App1
MatrizPontos[Pallet_1,Prdt_35BarPacking,1].XApp2Place=P1_35BarPacking_1_App2
MatrizPontos[Pallet_1,Prdt_35BarPacking,1].XPlace=P1_35BarPacking_1_Place
;ENDFOLD
;FOLD OffsetPlace
MatrizPontos[Pallet_1,Prdt_35BarPacking,1].OffsetPlace.X=0
MatrizPontos[Pallet_1,Prdt_35BarPacking,1].OffsetPlace.Y=0
MatrizPontos[Pallet_1,Prdt_35BarPacking,1].OffsetPlace.Z=0
MatrizPontos[Pallet_1,Prdt_35BarPacking,1].OffsetPlace.A=0
MatrizPontos[Pallet_1,Prdt_35BarPacking,1].OffsetPlace.B=0
MatrizPontos[Pallet_1,Prdt_35BarPacking,1].OffsetPlace.C=0
;ENDFOLD
;ENDFOLD

;FOLD PLACE 2
;FOLD PROPRIEDADES
MatrizPontos[Pallet_1,Prdt_35BarPacking,2].NumCaixas = 1
MatrizPontos[Pallet_1,Prdt_35BarPacking,2].PickOp = 2
MatrizPontos[Pallet_1,Prdt_35BarPacking,2].ConfGarraOp = 2
MatrizPontos[Pallet_1,Prdt_35BarPacking,2].FechaGarraOp = 0
MatrizPontos[Pallet_1,Prdt_35BarPacking,2].AbreGarraOp = 0
MatrizPontos[Pallet_1,Prdt_35BarPacking,2].SensoresCaixa = 12
MatrizPontos[Pallet_1,Prdt_35BarPacking,2].TravaGarra = False
MatrizPontos[Pallet_1,Prdt_35BarPacking,2].SkipGoHome = False
MatrizPontos[Pallet_1,Prdt_35BarPacking,2].SkipSobeRelAtual = False
MatrizPontos[Pallet_1,Prdt_35BarPacking,2].XApp1Place=P1_35BarPacking_2_App1
MatrizPontos[Pallet_1,Prdt_35BarPacking,2].XApp2Place=P1_35BarPacking_2_App2
MatrizPontos[Pallet_1,Prdt_35BarPacking,2].XPlace=P1_35BarPacking_2_Place
;ENDFOLD
;FOLD OffsetPlace
MatrizPontos[Pallet_1,Prdt_35BarPacking,2].OffsetPlace.X=0
MatrizPontos[Pallet_1,Prdt_35BarPacking,2].OffsetPlace.Y=0
MatrizPontos[Pallet_1,Prdt_35BarPacking,2].OffsetPlace.Z=0
MatrizPontos[Pallet_1,Prdt_35BarPacking,2].OffsetPlace.A=0
MatrizPontos[Pallet_1,Prdt_35BarPacking,2].OffsetPlace.B=0
MatrizPontos[Pallet_1,Prdt_35BarPacking,2].OffsetPlace.C=0
;ENDFOLD
;ENDFOLD

;FOLD PLACE 3
;FOLD PROPRIEDADES
MatrizPontos[Pallet_1,Prdt_35BarPacking,3].NumCaixas = 3
MatrizPontos[Pallet_1,Prdt_35BarPacking,3].PickOp = 2
MatrizPontos[Pallet_1,Prdt_35BarPacking,3].ConfGarraOp = 2
MatrizPontos[Pallet_1,Prdt_35BarPacking,3].FechaGarraOp = 0
MatrizPontos[Pallet_1,Prdt_35BarPacking,3].AbreGarraOp = 0
MatrizPontos[Pallet_1,Prdt_35BarPacking,3].SensoresCaixa = 123456
MatrizPontos[Pallet_1,Prdt_35BarPacking,3].TravaGarra = False
MatrizPontos[Pallet_1,Prdt_35BarPacking,3].SkipGoHome = False
MatrizPontos[Pallet_1,Prdt_35BarPacking,3].SkipSobeRelAtual = False
MatrizPontos[Pallet_1,Prdt_35BarPacking,3].XApp1Place=P1_35BarPacking_3_App1
MatrizPontos[Pallet_1,Prdt_35BarPacking,3].XApp2Place=P1_35BarPacking_3_App2
MatrizPontos[Pallet_1,Prdt_35BarPacking,3].XPlace=P1_35BarPacking_3_Place
;ENDFOLD
;FOLD OffsetPlace
MatrizPontos[Pallet_1,Prdt_35BarPacking,3].OffsetPlace.X=0
MatrizPontos[Pallet_1,Prdt_35BarPacking,3].OffsetPlace.Y=0
MatrizPontos[Pallet_1,Prdt_35BarPacking,3].OffsetPlace.Z=0
MatrizPontos[Pallet_1,Prdt_35BarPacking,3].OffsetPlace.A=0
MatrizPontos[Pallet_1,Prdt_35BarPacking,3].OffsetPlace.B=0
MatrizPontos[Pallet_1,Prdt_35BarPacking,3].OffsetPlace.C=0
;ENDFOLD
;ENDFOLD

;ENDFOLD
;ENDFOLD

;ENDFOLD
;FOLD PALLET 2
;FOLD Pallet 2 - Produto 1Aero
;FOLD LAYER 1: PLACE 1 ate 8
;FOLD PLACE 1
;FOLD PROPRIEDADES
MatrizPontos[Pallet_2,Prdt_1Aero,1].NumCaixas = 5
MatrizPontos[Pallet_2,Prdt_1Aero,1].PickOp = 7
MatrizPontos[Pallet_2,Prdt_1Aero,1].ConfGarraOp = 1
MatrizPontos[Pallet_2,Prdt_1Aero,1].FechaGarraOp = 0
MatrizPontos[Pallet_2,Prdt_1Aero,1].AbreGarraOp = 0
MatrizPontos[Pallet_2,Prdt_1Aero,1].SensoresCaixa = 12345
MatrizPontos[Pallet_2,Prdt_1Aero,1].TravaGarra = False
MatrizPontos[Pallet_2,Prdt_1Aero,1].SkipGoHome = False
MatrizPontos[Pallet_2,Prdt_1Aero,1].SkipSobeRelAtual = False
MatrizPontos[Pallet_2,Prdt_1Aero,1].XApp1Place=P2_1Aero_1_App1
MatrizPontos[Pallet_2,Prdt_1Aero,1].XApp2Place=P2_1Aero_1_App2
MatrizPontos[Pallet_2,Prdt_1Aero,1].XPlace=P2_1Aero_1_Place
;ENDFOLD
;FOLD OffsetPlace
MatrizPontos[Pallet_2,Prdt_1Aero,1].OffsetPlace.X=0
MatrizPontos[Pallet_2,Prdt_1Aero,1].OffsetPlace.Y=0
MatrizPontos[Pallet_2,Prdt_1Aero,1].OffsetPlace.Z=0
MatrizPontos[Pallet_2,Prdt_1Aero,1].OffsetPlace.A=0
MatrizPontos[Pallet_2,Prdt_1Aero,1].OffsetPlace.B=0
MatrizPontos[Pallet_2,Prdt_1Aero,1].OffsetPlace.C=0
;ENDFOLD
;ENDFOLD

;FOLD PLACE 2
;FOLD PROPRIEDADES
MatrizPontos[Pallet_2,Prdt_1Aero,2].NumCaixas = 5
MatrizPontos[Pallet_2,Prdt_1Aero,2].PickOp = 7
MatrizPontos[Pallet_2,Prdt_1Aero,2].ConfGarraOp = 1
MatrizPontos[Pallet_2,Prdt_1Aero,2].FechaGarraOp = 0
MatrizPontos[Pallet_2,Prdt_1Aero,2].AbreGarraOp = 0
MatrizPontos[Pallet_2,Prdt_1Aero,2].SensoresCaixa = 12345
MatrizPontos[Pallet_2,Prdt_1Aero,2].TravaGarra = False
MatrizPontos[Pallet_2,Prdt_1Aero,2].SkipGoHome = False
MatrizPontos[Pallet_2,Prdt_1Aero,2].SkipSobeRelAtual = False
MatrizPontos[Pallet_2,Prdt_1Aero,2].XApp1Place=P2_1Aero_2_App1
MatrizPontos[Pallet_2,Prdt_1Aero,2].XApp2Place=P2_1Aero_2_App2
MatrizPontos[Pallet_2,Prdt_1Aero,2].XPlace=P2_1Aero_2_Place
;ENDFOLD
;FOLD OffsetPlace
MatrizPontos[Pallet_2,Prdt_1Aero,2].OffsetPlace.X=0
MatrizPontos[Pallet_2,Prdt_1Aero,2].OffsetPlace.Y=0
MatrizPontos[Pallet_2,Prdt_1Aero,2].OffsetPlace.Z=0
MatrizPontos[Pallet_2,Prdt_1Aero,2].OffsetPlace.A=0
MatrizPontos[Pallet_2,Prdt_1Aero,2].OffsetPlace.B=0
MatrizPontos[Pallet_2,Prdt_1Aero,2].OffsetPlace.C=0
;ENDFOLD
;ENDFOLD

;FOLD PLACE 3
;FOLD PROPRIEDADES
MatrizPontos[Pallet_2,Prdt_1Aero,3].NumCaixas = 5
MatrizPontos[Pallet_2,Prdt_1Aero,3].PickOp = 7
MatrizPontos[Pallet_2,Prdt_1Aero,3].ConfGarraOp = 1
MatrizPontos[Pallet_2,Prdt_1Aero,3].FechaGarraOp = 0
MatrizPontos[Pallet_2,Prdt_1Aero,3].AbreGarraOp = 0
MatrizPontos[Pallet_2,Prdt_1Aero,3].SensoresCaixa = 12345
MatrizPontos[Pallet_2,Prdt_1Aero,3].TravaGarra = False
MatrizPontos[Pallet_2,Prdt_1Aero,3].SkipGoHome = False
MatrizPontos[Pallet_2,Prdt_1Aero,3].SkipSobeRelAtual = False
MatrizPontos[Pallet_2,Prdt_1Aero,3].XApp1Place=P2_1Aero_3_App1
MatrizPontos[Pallet_2,Prdt_1Aero,3].XApp2Place=P2_1Aero_3_App2
MatrizPontos[Pallet_2,Prdt_1Aero,3].XPlace=P2_1Aero_3_Place
;ENDFOLD
;FOLD OffsetPlace
MatrizPontos[Pallet_2,Prdt_1Aero,3].OffsetPlace.X=0
MatrizPontos[Pallet_2,Prdt_1Aero,3].OffsetPlace.Y=0
MatrizPontos[Pallet_2,Prdt_1Aero,3].OffsetPlace.Z=0
MatrizPontos[Pallet_2,Prdt_1Aero,3].OffsetPlace.A=0
MatrizPontos[Pallet_2,Prdt_1Aero,3].OffsetPlace.B=0
MatrizPontos[Pallet_2,Prdt_1Aero,3].OffsetPlace.C=0
;ENDFOLD
;ENDFOLD

;FOLD PLACE 4
;FOLD PROPRIEDADES
MatrizPontos[Pallet_2,Prdt_1Aero,4].NumCaixas = 5
MatrizPontos[Pallet_2,Prdt_1Aero,4].PickOp = 7
MatrizPontos[Pallet_2,Prdt_1Aero,4].ConfGarraOp = 1
MatrizPontos[Pallet_2,Prdt_1Aero,4].FechaGarraOp = 0
MatrizPontos[Pallet_2,Prdt_1Aero,4].AbreGarraOp = 2
MatrizPontos[Pallet_2,Prdt_1Aero,4].SensoresCaixa = 1
MatrizPontos[Pallet_2,Prdt_1Aero,4].TravaGarra = False
MatrizPontos[Pallet_2,Prdt_1Aero,4].SkipGoHome = True
MatrizPontos[Pallet_2,Prdt_1Aero,4].SkipSobeRelAtual = True
MatrizPontos[Pallet_2,Prdt_1Aero,4].XApp1Place=P2_1Aero_4_App1
MatrizPontos[Pallet_2,Prdt_1Aero,4].XApp2Place=P2_1Aero_4_App2
MatrizPontos[Pallet_2,Prdt_1Aero,4].XPlace=P2_1Aero_4_Place
;ENDFOLD
;FOLD OffsetPlace
MatrizPontos[Pallet_2,Prdt_1Aero,4].OffsetPlace.X=0
MatrizPontos[Pallet_2,Prdt_1Aero,4].OffsetPlace.Y=0
MatrizPontos[Pallet_2,Prdt_1Aero,4].OffsetPlace.Z=0
MatrizPontos[Pallet_2,Prdt_1Aero,4].OffsetPlace.A=0
MatrizPontos[Pallet_2,Prdt_1Aero,4].OffsetPlace.B=0
MatrizPontos[Pallet_2,Prdt_1Aero,4].OffsetPlace.C=0
;ENDFOLD
;ENDFOLD

;FOLD PLACE 5
;FOLD PROPRIEDADES
MatrizPontos[Pallet_2,Prdt_1Aero,5].NumCaixas = 5
MatrizPontos[Pallet_2,Prdt_1Aero,5].PickOp = 7
MatrizPontos[Pallet_2,Prdt_1Aero,5].ConfGarraOp = 1
MatrizPontos[Pallet_2,Prdt_1Aero,5].FechaGarraOp = 0
MatrizPontos[Pallet_2,Prdt_1Aero,5].AbreGarraOp = 3
MatrizPontos[Pallet_2,Prdt_1Aero,5].SensoresCaixa = 2
MatrizPontos[Pallet_2,Prdt_1Aero,5].TravaGarra = False
MatrizPontos[Pallet_2,Prdt_1Aero,5].SkipGoHome = True
MatrizPontos[Pallet_2,Prdt_1Aero,5].SkipSobeRelAtual = True
MatrizPontos[Pallet_2,Prdt_1Aero,5].XApp1Place=P2_1Aero_5_App1
MatrizPontos[Pallet_2,Prdt_1Aero,5].XApp2Place=P2_1Aero_5_App2
MatrizPontos[Pallet_2,Prdt_1Aero,5].XPlace=P2_1Aero_5_Place
;ENDFOLD
;FOLD OffsetPlace
MatrizPontos[Pallet_2,Prdt_1Aero,5].OffsetPlace.X=0
MatrizPontos[Pallet_2,Prdt_1Aero,5].OffsetPlace.Y=0
MatrizPontos[Pallet_2,Prdt_1Aero,5].OffsetPlace.Z=0
MatrizPontos[Pallet_2,Prdt_1Aero,5].OffsetPlace.A=0
MatrizPontos[Pallet_2,Prdt_1Aero,5].OffsetPlace.B=0
MatrizPontos[Pallet_2,Prdt_1Aero,5].OffsetPlace.C=0
;ENDFOLD
;ENDFOLD

;FOLD PLACE 6
;FOLD PROPRIEDADES
MatrizPontos[Pallet_2,Prdt_1Aero,6].NumCaixas = 5
MatrizPontos[Pallet_2,Prdt_1Aero,6].PickOp = 7
MatrizPontos[Pallet_2,Prdt_1Aero,6].ConfGarraOp = 1
MatrizPontos[Pallet_2,Prdt_1Aero,6].FechaGarraOp = 0
MatrizPontos[Pallet_2,Prdt_1Aero,6].AbreGarraOp = 4
MatrizPontos[Pallet_2,Prdt_1Aero,6].SensoresCaixa = 3
MatrizPontos[Pallet_2,Prdt_1Aero,6].TravaGarra = False
MatrizPontos[Pallet_2,Prdt_1Aero,6].SkipGoHome = True
MatrizPontos[Pallet_2,Prdt_1Aero,6].SkipSobeRelAtual = True
MatrizPontos[Pallet_2,Prdt_1Aero,6].XApp1Place=P2_1Aero_6_App1
MatrizPontos[Pallet_2,Prdt_1Aero,6].XApp2Place=P2_1Aero_6_App2
MatrizPontos[Pallet_2,Prdt_1Aero,6].XPlace=P2_1Aero_6_Place
;ENDFOLD
;FOLD OffsetPlace
MatrizPontos[Pallet_2,Prdt_1Aero,6].OffsetPlace.X=0
MatrizPontos[Pallet_2,Prdt_1Aero,6].OffsetPlace.Y=0
MatrizPontos[Pallet_2,Prdt_1Aero,6].OffsetPlace.Z=0
MatrizPontos[Pallet_2,Prdt_1Aero,6].OffsetPlace.A=0
MatrizPontos[Pallet_2,Prdt_1Aero,6].OffsetPlace.B=0
MatrizPontos[Pallet_2,Prdt_1Aero,6].OffsetPlace.C=0
;ENDFOLD
;ENDFOLD

;FOLD PLACE 7
;FOLD PROPRIEDADES
MatrizPontos[Pallet_2,Prdt_1Aero,7].NumCaixas = 5
MatrizPontos[Pallet_2,Prdt_1Aero,7].PickOp = 7
MatrizPontos[Pallet_2,Prdt_1Aero,7].ConfGarraOp = 1
MatrizPontos[Pallet_2,Prdt_1Aero,7].FechaGarraOp = 0
MatrizPontos[Pallet_2,Prdt_1Aero,7].AbreGarraOp = 5
MatrizPontos[Pallet_2,Prdt_1Aero,7].SensoresCaixa = 4
MatrizPontos[Pallet_2,Prdt_1Aero,7].TravaGarra = False
MatrizPontos[Pallet_2,Prdt_1Aero,7].SkipGoHome = True
MatrizPontos[Pallet_2,Prdt_1Aero,7].SkipSobeRelAtual = True
MatrizPontos[Pallet_2,Prdt_1Aero,7].XApp1Place=P2_1Aero_7_App1
MatrizPontos[Pallet_2,Prdt_1Aero,7].XApp2Place=P2_1Aero_7_App2
MatrizPontos[Pallet_2,Prdt_1Aero,7].XPlace=P2_1Aero_7_Place
;ENDFOLD
;FOLD OffsetPlace
MatrizPontos[Pallet_2,Prdt_1Aero,7].OffsetPlace.X=0
MatrizPontos[Pallet_2,Prdt_1Aero,7].OffsetPlace.Y=0
MatrizPontos[Pallet_2,Prdt_1Aero,7].OffsetPlace.Z=0
MatrizPontos[Pallet_2,Prdt_1Aero,7].OffsetPlace.A=0
MatrizPontos[Pallet_2,Prdt_1Aero,7].OffsetPlace.B=0
MatrizPontos[Pallet_2,Prdt_1Aero,7].OffsetPlace.C=0
;ENDFOLD
;ENDFOLD

;FOLD PLACE 8
;FOLD PROPRIEDADES
MatrizPontos[Pallet_2,Prdt_1Aero,8].NumCaixas = 5
MatrizPontos[Pallet_2,Prdt_1Aero,8].PickOp = 7
MatrizPontos[Pallet_2,Prdt_1Aero,8].ConfGarraOp = 1
MatrizPontos[Pallet_2,Prdt_1Aero,8].FechaGarraOp = 0
MatrizPontos[Pallet_2,Prdt_1Aero,8].AbreGarraOp = 6
MatrizPontos[Pallet_2,Prdt_1Aero,8].SensoresCaixa = 5
MatrizPontos[Pallet_2,Prdt_1Aero,8].TravaGarra = False
MatrizPontos[Pallet_2,Prdt_1Aero,8].SkipGoHome = True
MatrizPontos[Pallet_2,Prdt_1Aero,8].SkipSobeRelAtual = True
MatrizPontos[Pallet_2,Prdt_1Aero,8].XApp1Place=P2_1Aero_8_App1
MatrizPontos[Pallet_2,Prdt_1Aero,8].XApp2Place=P2_1Aero_8_App2
MatrizPontos[Pallet_2,Prdt_1Aero,8].XPlace=P2_1Aero_8_Place
;ENDFOLD
;FOLD OffsetPlace
MatrizPontos[Pallet_2,Prdt_1Aero,8].OffsetPlace.X=0
MatrizPontos[Pallet_2,Prdt_1Aero,8].OffsetPlace.Y=0
MatrizPontos[Pallet_2,Prdt_1Aero,8].OffsetPlace.Z=0
MatrizPontos[Pallet_2,Prdt_1Aero,8].OffsetPlace.A=0
MatrizPontos[Pallet_2,Prdt_1Aero,8].OffsetPlace.B=0
MatrizPontos[Pallet_2,Prdt_1Aero,8].OffsetPlace.C=0
;ENDFOLD
;ENDFOLD

;ENDFOLD
;FOLD LAYER 2: PLACE 9 ate 16
;FOLD PLACE 9
;FOLD PROPRIEDADES
MatrizPontos[Pallet_2,Prdt_1Aero,9].NumCaixas = 5
MatrizPontos[Pallet_2,Prdt_1Aero,9].PickOp = 7
MatrizPontos[Pallet_2,Prdt_1Aero,9].ConfGarraOp = 1
MatrizPontos[Pallet_2,Prdt_1Aero,9].FechaGarraOp = 0
MatrizPontos[Pallet_2,Prdt_1Aero,9].AbreGarraOp = 2
MatrizPontos[Pallet_2,Prdt_1Aero,9].SensoresCaixa = 1
MatrizPontos[Pallet_2,Prdt_1Aero,9].TravaGarra = False
MatrizPontos[Pallet_2,Prdt_1Aero,9].SkipGoHome = True
MatrizPontos[Pallet_2,Prdt_1Aero,9].SkipSobeRelAtual = True
MatrizPontos[Pallet_2,Prdt_1Aero,9].XApp1Place=P2_1Aero_9_App1
MatrizPontos[Pallet_2,Prdt_1Aero,9].XApp2Place=P2_1Aero_9_App2
MatrizPontos[Pallet_2,Prdt_1Aero,9].XPlace=P2_1Aero_9_Place
;ENDFOLD
;FOLD OffsetPlace
MatrizPontos[Pallet_2,Prdt_1Aero,9].OffsetPlace.X=0
MatrizPontos[Pallet_2,Prdt_1Aero,9].OffsetPlace.Y=0
MatrizPontos[Pallet_2,Prdt_1Aero,9].OffsetPlace.Z=0
MatrizPontos[Pallet_2,Prdt_1Aero,9].OffsetPlace.A=0
MatrizPontos[Pallet_2,Prdt_1Aero,9].OffsetPlace.B=0
MatrizPontos[Pallet_2,Prdt_1Aero,9].OffsetPlace.C=0
;ENDFOLD
;ENDFOLD

;FOLD PLACE 10
;FOLD PROPRIEDADES
MatrizPontos[Pallet_2,Prdt_1Aero,10].NumCaixas = 5
MatrizPontos[Pallet_2,Prdt_1Aero,10].PickOp = 7
MatrizPontos[Pallet_2,Prdt_1Aero,10].ConfGarraOp = 1
MatrizPontos[Pallet_2,Prdt_1Aero,10].FechaGarraOp = 0
MatrizPontos[Pallet_2,Prdt_1Aero,10].AbreGarraOp = 3
MatrizPontos[Pallet_2,Prdt_1Aero,10].SensoresCaixa = 2
MatrizPontos[Pallet_2,Prdt_1Aero,10].TravaGarra = False
MatrizPontos[Pallet_2,Prdt_1Aero,10].SkipGoHome = True
MatrizPontos[Pallet_2,Prdt_1Aero,10].SkipSobeRelAtual = True
MatrizPontos[Pallet_2,Prdt_1Aero,10].XApp1Place=P2_1Aero_10_App1
MatrizPontos[Pallet_2,Prdt_1Aero,10].XApp2Place=P2_1Aero_10_App2
MatrizPontos[Pallet_2,Prdt_1Aero,10].XPlace=P2_1Aero_10_Place
;ENDFOLD
;FOLD OffsetPlace
MatrizPontos[Pallet_2,Prdt_1Aero,10].OffsetPlace.X=0
MatrizPontos[Pallet_2,Prdt_1Aero,10].OffsetPlace.Y=0
MatrizPontos[Pallet_2,Prdt_1Aero,10].OffsetPlace.Z=0
MatrizPontos[Pallet_2,Prdt_1Aero,10].OffsetPlace.A=0
MatrizPontos[Pallet_2,Prdt_1Aero,10].OffsetPlace.B=0
MatrizPontos[Pallet_2,Prdt_1Aero,10].OffsetPlace.C=0
;ENDFOLD
;ENDFOLD

;FOLD PLACE 11
;FOLD PROPRIEDADES
MatrizPontos[Pallet_2,Prdt_1Aero,11].NumCaixas = 5
MatrizPontos[Pallet_2,Prdt_1Aero,11].PickOp = 7
MatrizPontos[Pallet_2,Prdt_1Aero,11].ConfGarraOp = 1
MatrizPontos[Pallet_2,Prdt_1Aero,11].FechaGarraOp = 0
MatrizPontos[Pallet_2,Prdt_1Aero,11].AbreGarraOp = 4
MatrizPontos[Pallet_2,Prdt_1Aero,11].SensoresCaixa = 3
MatrizPontos[Pallet_2,Prdt_1Aero,11].TravaGarra = False
MatrizPontos[Pallet_2,Prdt_1Aero,11].SkipGoHome = True
MatrizPontos[Pallet_2,Prdt_1Aero,11].SkipSobeRelAtual = True
MatrizPontos[Pallet_2,Prdt_1Aero,11].XApp1Place=P2_1Aero_11_App1
MatrizPontos[Pallet_2,Prdt_1Aero,11].XApp2Place=P2_1Aero_11_App2
MatrizPontos[Pallet_2,Prdt_1Aero,11].XPlace=P2_1Aero_11_Place
;ENDFOLD
;FOLD OffsetPlace
MatrizPontos[Pallet_2,Prdt_1Aero,11].OffsetPlace.X=0
MatrizPontos[Pallet_2,Prdt_1Aero,11].OffsetPlace.Y=0
MatrizPontos[Pallet_2,Prdt_1Aero,11].OffsetPlace.Z=0
MatrizPontos[Pallet_2,Prdt_1Aero,11].OffsetPlace.A=0
MatrizPontos[Pallet_2,Prdt_1Aero,11].OffsetPlace.B=0
MatrizPontos[Pallet_2,Prdt_1Aero,11].OffsetPlace.C=0
;ENDFOLD
;ENDFOLD

;FOLD PLACE 12
;FOLD PROPRIEDADES
MatrizPontos[Pallet_2,Prdt_1Aero,12].NumCaixas = 5
MatrizPontos[Pallet_2,Prdt_1Aero,12].PickOp = 7
MatrizPontos[Pallet_2,Prdt_1Aero,12].ConfGarraOp = 1
MatrizPontos[Pallet_2,Prdt_1Aero,12].FechaGarraOp = 0
MatrizPontos[Pallet_2,Prdt_1Aero,12].AbreGarraOp = 5
MatrizPontos[Pallet_2,Prdt_1Aero,12].SensoresCaixa = 4
MatrizPontos[Pallet_2,Prdt_1Aero,12].TravaGarra = False
MatrizPontos[Pallet_2,Prdt_1Aero,12].SkipGoHome = True
MatrizPontos[Pallet_2,Prdt_1Aero,12].SkipSobeRelAtual = True
MatrizPontos[Pallet_2,Prdt_1Aero,12].XApp1Place=P2_1Aero_12_App1
MatrizPontos[Pallet_2,Prdt_1Aero,12].XApp2Place=P2_1Aero_12_App2
MatrizPontos[Pallet_2,Prdt_1Aero,12].XPlace=P2_1Aero_12_Place
;ENDFOLD
;FOLD OffsetPlace
MatrizPontos[Pallet_2,Prdt_1Aero,12].OffsetPlace.X=0
MatrizPontos[Pallet_2,Prdt_1Aero,12].OffsetPlace.Y=0
MatrizPontos[Pallet_2,Prdt_1Aero,12].OffsetPlace.Z=0
MatrizPontos[Pallet_2,Prdt_1Aero,12].OffsetPlace.A=0
MatrizPontos[Pallet_2,Prdt_1Aero,12].OffsetPlace.B=0
MatrizPontos[Pallet_2,Prdt_1Aero,12].OffsetPlace.C=0
;ENDFOLD
;ENDFOLD

;FOLD PLACE 13
;FOLD PROPRIEDADES
MatrizPontos[Pallet_2,Prdt_1Aero,13].NumCaixas = 5
MatrizPontos[Pallet_2,Prdt_1Aero,13].PickOp = 7
MatrizPontos[Pallet_2,Prdt_1Aero,13].ConfGarraOp = 1
MatrizPontos[Pallet_2,Prdt_1Aero,13].FechaGarraOp = 0
MatrizPontos[Pallet_2,Prdt_1Aero,13].AbreGarraOp = 6
MatrizPontos[Pallet_2,Prdt_1Aero,13].SensoresCaixa = 5
MatrizPontos[Pallet_2,Prdt_1Aero,13].TravaGarra = False
MatrizPontos[Pallet_2,Prdt_1Aero,13].SkipGoHome = True
MatrizPontos[Pallet_2,Prdt_1Aero,13].SkipSobeRelAtual = True
MatrizPontos[Pallet_2,Prdt_1Aero,13].XApp1Place=P2_1Aero_13_App1
MatrizPontos[Pallet_2,Prdt_1Aero,13].XApp2Place=P2_1Aero_13_App2
MatrizPontos[Pallet_2,Prdt_1Aero,13].XPlace=P2_1Aero_13_Place
;ENDFOLD
;FOLD OffsetPlace
MatrizPontos[Pallet_2,Prdt_1Aero,13].OffsetPlace.X=0
MatrizPontos[Pallet_2,Prdt_1Aero,13].OffsetPlace.Y=0
MatrizPontos[Pallet_2,Prdt_1Aero,13].OffsetPlace.Z=0
MatrizPontos[Pallet_2,Prdt_1Aero,13].OffsetPlace.A=0
MatrizPontos[Pallet_2,Prdt_1Aero,13].OffsetPlace.B=0
MatrizPontos[Pallet_2,Prdt_1Aero,13].OffsetPlace.C=0
;ENDFOLD
;ENDFOLD

;FOLD PLACE 14
;FOLD PROPRIEDADES
MatrizPontos[Pallet_2,Prdt_1Aero,14].NumCaixas = 5
MatrizPontos[Pallet_2,Prdt_1Aero,14].PickOp = 7
MatrizPontos[Pallet_2,Prdt_1Aero,14].ConfGarraOp = 1
MatrizPontos[Pallet_2,Prdt_1Aero,14].FechaGarraOp = 0
MatrizPontos[Pallet_2,Prdt_1Aero,14].AbreGarraOp = 0
MatrizPontos[Pallet_2,Prdt_1Aero,14].SensoresCaixa = 12345
MatrizPontos[Pallet_2,Prdt_1Aero,14].TravaGarra = False
MatrizPontos[Pallet_2,Prdt_1Aero,14].SkipGoHome = False
MatrizPontos[Pallet_2,Prdt_1Aero,14].SkipSobeRelAtual = False
MatrizPontos[Pallet_2,Prdt_1Aero,14].XApp1Place=P2_1Aero_14_App1
MatrizPontos[Pallet_2,Prdt_1Aero,14].XApp2Place=P2_1Aero_14_App2
MatrizPontos[Pallet_2,Prdt_1Aero,14].XPlace=P2_1Aero_14_Place
;ENDFOLD
;FOLD OffsetPlace
MatrizPontos[Pallet_2,Prdt_1Aero,14].OffsetPlace.X=0
MatrizPontos[Pallet_2,Prdt_1Aero,14].OffsetPlace.Y=0
MatrizPontos[Pallet_2,Prdt_1Aero,14].OffsetPlace.Z=0
MatrizPontos[Pallet_2,Prdt_1Aero,14].OffsetPlace.A=0
MatrizPontos[Pallet_2,Prdt_1Aero,14].OffsetPlace.B=0
MatrizPontos[Pallet_2,Prdt_1Aero,14].OffsetPlace.C=0
;ENDFOLD
;ENDFOLD

;FOLD PLACE 15
;FOLD PROPRIEDADES
MatrizPontos[Pallet_2,Prdt_1Aero,15].NumCaixas = 5
MatrizPontos[Pallet_2,Prdt_1Aero,15].PickOp = 7
MatrizPontos[Pallet_2,Prdt_1Aero,15].ConfGarraOp = 1
MatrizPontos[Pallet_2,Prdt_1Aero,15].FechaGarraOp = 0
MatrizPontos[Pallet_2,Prdt_1Aero,15].AbreGarraOp = 0
MatrizPontos[Pallet_2,Prdt_1Aero,15].SensoresCaixa = 12345
MatrizPontos[Pallet_2,Prdt_1Aero,15].TravaGarra = False
MatrizPontos[Pallet_2,Prdt_1Aero,15].SkipGoHome = False
MatrizPontos[Pallet_2,Prdt_1Aero,15].SkipSobeRelAtual = False
MatrizPontos[Pallet_2,Prdt_1Aero,15].XApp1Place=P2_1Aero_15_App1
MatrizPontos[Pallet_2,Prdt_1Aero,15].XApp2Place=P2_1Aero_15_App2
MatrizPontos[Pallet_2,Prdt_1Aero,15].XPlace=P2_1Aero_15_Place
;ENDFOLD
;FOLD OffsetPlace
MatrizPontos[Pallet_2,Prdt_1Aero,15].OffsetPlace.X=0
MatrizPontos[Pallet_2,Prdt_1Aero,15].OffsetPlace.Y=0
MatrizPontos[Pallet_2,Prdt_1Aero,15].OffsetPlace.Z=0
MatrizPontos[Pallet_2,Prdt_1Aero,15].OffsetPlace.A=0
MatrizPontos[Pallet_2,Prdt_1Aero,15].OffsetPlace.B=0
MatrizPontos[Pallet_2,Prdt_1Aero,15].OffsetPlace.C=0
;ENDFOLD
;ENDFOLD

;FOLD PLACE 16
;FOLD PROPRIEDADES
MatrizPontos[Pallet_2,Prdt_1Aero,16].NumCaixas = 5
MatrizPontos[Pallet_2,Prdt_1Aero,16].PickOp = 7
MatrizPontos[Pallet_2,Prdt_1Aero,16].ConfGarraOp = 1
MatrizPontos[Pallet_2,Prdt_1Aero,16].FechaGarraOp = 0
MatrizPontos[Pallet_2,Prdt_1Aero,16].AbreGarraOp = 0
MatrizPontos[Pallet_2,Prdt_1Aero,16].SensoresCaixa = 12345
MatrizPontos[Pallet_2,Prdt_1Aero,16].TravaGarra = False
MatrizPontos[Pallet_2,Prdt_1Aero,16].SkipGoHome = False
MatrizPontos[Pallet_2,Prdt_1Aero,16].SkipSobeRelAtual = False
MatrizPontos[Pallet_2,Prdt_1Aero,16].XApp1Place=P2_1Aero_16_App1
MatrizPontos[Pallet_2,Prdt_1Aero,16].XApp2Place=P2_1Aero_16_App2
MatrizPontos[Pallet_2,Prdt_1Aero,16].XPlace=P2_1Aero_16_Place
;ENDFOLD
;FOLD OffsetPlace
MatrizPontos[Pallet_2,Prdt_1Aero,16].OffsetPlace.X=0
MatrizPontos[Pallet_2,Prdt_1Aero,16].OffsetPlace.Y=0
MatrizPontos[Pallet_2,Prdt_1Aero,16].OffsetPlace.Z=0
MatrizPontos[Pallet_2,Prdt_1Aero,16].OffsetPlace.A=0
MatrizPontos[Pallet_2,Prdt_1Aero,16].OffsetPlace.B=0
MatrizPontos[Pallet_2,Prdt_1Aero,16].OffsetPlace.C=0
;ENDFOLD
;ENDFOLD

;ENDFOLD
;ENDFOLD

;FOLD Pallet 2 - Produto 2Aero
;FOLD LAYER 1: PLACE 1 ate 3
;FOLD PLACE 1
;FOLD PROPRIEDADES
MatrizPontos[Pallet_2,Prdt_2Aero,1].NumCaixas = 4
MatrizPontos[Pallet_2,Prdt_2Aero,1].PickOp = 1
MatrizPontos[Pallet_2,Prdt_2Aero,1].ConfGarraOp = 0
MatrizPontos[Pallet_2,Prdt_2Aero,1].FechaGarraOp = 0
MatrizPontos[Pallet_2,Prdt_2Aero,1].AbreGarraOp = 0
MatrizPontos[Pallet_2,Prdt_2Aero,1].SensoresCaixa = 123456
MatrizPontos[Pallet_2,Prdt_2Aero,1].TravaGarra = False
MatrizPontos[Pallet_2,Prdt_2Aero,1].SkipGoHome = False
MatrizPontos[Pallet_2,Prdt_2Aero,1].SkipSobeRelAtual = False
MatrizPontos[Pallet_2,Prdt_2Aero,1].XApp1Place=P2_2Aero_1_App1
MatrizPontos[Pallet_2,Prdt_2Aero,1].XApp2Place=P2_2Aero_1_App2
MatrizPontos[Pallet_2,Prdt_2Aero,1].XPlace=P2_2Aero_1_Place
;ENDFOLD
;FOLD OffsetPlace
MatrizPontos[Pallet_2,Prdt_2Aero,1].OffsetPlace.X=0
MatrizPontos[Pallet_2,Prdt_2Aero,1].OffsetPlace.Y=0
MatrizPontos[Pallet_2,Prdt_2Aero,1].OffsetPlace.Z=0
MatrizPontos[Pallet_2,Prdt_2Aero,1].OffsetPlace.A=0
MatrizPontos[Pallet_2,Prdt_2Aero,1].OffsetPlace.B=0
MatrizPontos[Pallet_2,Prdt_2Aero,1].OffsetPlace.C=0
;ENDFOLD
;ENDFOLD

;FOLD PLACE 2
;FOLD PROPRIEDADES
MatrizPontos[Pallet_2,Prdt_2Aero,2].NumCaixas = 4
MatrizPontos[Pallet_2,Prdt_2Aero,2].PickOp = 1
MatrizPontos[Pallet_2,Prdt_2Aero,2].ConfGarraOp = 0
MatrizPontos[Pallet_2,Prdt_2Aero,2].FechaGarraOp = 0
MatrizPontos[Pallet_2,Prdt_2Aero,2].AbreGarraOp = 0
MatrizPontos[Pallet_2,Prdt_2Aero,2].SensoresCaixa = 123456
MatrizPontos[Pallet_2,Prdt_2Aero,2].TravaGarra = False
MatrizPontos[Pallet_2,Prdt_2Aero,2].SkipGoHome = False
MatrizPontos[Pallet_2,Prdt_2Aero,2].SkipSobeRelAtual = False
MatrizPontos[Pallet_2,Prdt_2Aero,2].XApp1Place=P2_2Aero_2_App1
MatrizPontos[Pallet_2,Prdt_2Aero,2].XApp2Place=P2_2Aero_2_App2
MatrizPontos[Pallet_2,Prdt_2Aero,2].XPlace=P2_2Aero_2_Place
;ENDFOLD
;FOLD OffsetPlace
MatrizPontos[Pallet_2,Prdt_2Aero,2].OffsetPlace.X=0
MatrizPontos[Pallet_2,Prdt_2Aero,2].OffsetPlace.Y=0
MatrizPontos[Pallet_2,Prdt_2Aero,2].OffsetPlace.Z=0
MatrizPontos[Pallet_2,Prdt_2Aero,2].OffsetPlace.A=0
MatrizPontos[Pallet_2,Prdt_2Aero,2].OffsetPlace.B=0
MatrizPontos[Pallet_2,Prdt_2Aero,2].OffsetPlace.C=0
;ENDFOLD
;ENDFOLD

;FOLD PLACE 3
;FOLD PROPRIEDADES
MatrizPontos[Pallet_2,Prdt_2Aero,3].NumCaixas = 4
MatrizPontos[Pallet_2,Prdt_2Aero,3].PickOp = 1
MatrizPontos[Pallet_2,Prdt_2Aero,3].ConfGarraOp = 0
MatrizPontos[Pallet_2,Prdt_2Aero,3].FechaGarraOp = 0
MatrizPontos[Pallet_2,Prdt_2Aero,3].AbreGarraOp = 0
MatrizPontos[Pallet_2,Prdt_2Aero,3].SensoresCaixa = 123456
MatrizPontos[Pallet_2,Prdt_2Aero,3].TravaGarra = False
MatrizPontos[Pallet_2,Prdt_2Aero,3].SkipGoHome = False
MatrizPontos[Pallet_2,Prdt_2Aero,3].SkipSobeRelAtual = False
MatrizPontos[Pallet_2,Prdt_2Aero,3].XApp1Place=P2_2Aero_3_App1
MatrizPontos[Pallet_2,Prdt_2Aero,3].XApp2Place=P2_2Aero_3_App2
MatrizPontos[Pallet_2,Prdt_2Aero,3].XPlace=P2_2Aero_3_Place
;ENDFOLD
;FOLD OffsetPlace
MatrizPontos[Pallet_2,Prdt_2Aero,3].OffsetPlace.X=0
MatrizPontos[Pallet_2,Prdt_2Aero,3].OffsetPlace.Y=0
MatrizPontos[Pallet_2,Prdt_2Aero,3].OffsetPlace.Z=0
MatrizPontos[Pallet_2,Prdt_2Aero,3].OffsetPlace.A=0
MatrizPontos[Pallet_2,Prdt_2Aero,3].OffsetPlace.B=0
MatrizPontos[Pallet_2,Prdt_2Aero,3].OffsetPlace.C=0
;ENDFOLD
;ENDFOLD

;ENDFOLD
;ENDFOLD

;FOLD Pallet 2 - Produto 5Aero
;FOLD LAYER 1: PLACE 1 ate 3
;FOLD PLACE 1
;FOLD PROPRIEDADES
MatrizPontos[Pallet_2,Prdt_5Aero,1].NumCaixas = 3
MatrizPontos[Pallet_2,Prdt_5Aero,1].PickOp = 1
MatrizPontos[Pallet_2,Prdt_5Aero,1].ConfGarraOp = 0
MatrizPontos[Pallet_2,Prdt_5Aero,1].FechaGarraOp = 0
MatrizPontos[Pallet_2,Prdt_5Aero,1].AbreGarraOp = 0
MatrizPontos[Pallet_2,Prdt_5Aero,1].SensoresCaixa = 12345
MatrizPontos[Pallet_2,Prdt_5Aero,1].TravaGarra = False
MatrizPontos[Pallet_2,Prdt_5Aero,1].SkipGoHome = False
MatrizPontos[Pallet_2,Prdt_5Aero,1].SkipSobeRelAtual = False
MatrizPontos[Pallet_2,Prdt_5Aero,1].XApp1Place=P2_5Aero_1_App1
MatrizPontos[Pallet_2,Prdt_5Aero,1].XApp2Place=P2_5Aero_1_App2
MatrizPontos[Pallet_2,Prdt_5Aero,1].XPlace=P2_5Aero_1_Place
;ENDFOLD
;FOLD OffsetPlace
MatrizPontos[Pallet_2,Prdt_5Aero,1].OffsetPlace.X=0
MatrizPontos[Pallet_2,Prdt_5Aero,1].OffsetPlace.Y=0
MatrizPontos[Pallet_2,Prdt_5Aero,1].OffsetPlace.Z=0
MatrizPontos[Pallet_2,Prdt_5Aero,1].OffsetPlace.A=0
MatrizPontos[Pallet_2,Prdt_5Aero,1].OffsetPlace.B=0
MatrizPontos[Pallet_2,Prdt_5Aero,1].OffsetPlace.C=0
;ENDFOLD
;ENDFOLD

;FOLD PLACE 2
;FOLD PROPRIEDADES
MatrizPontos[Pallet_2,Prdt_5Aero,2].NumCaixas = 3
MatrizPontos[Pallet_2,Prdt_5Aero,2].PickOp = 1
MatrizPontos[Pallet_2,Prdt_5Aero,2].ConfGarraOp = 0
MatrizPontos[Pallet_2,Prdt_5Aero,2].FechaGarraOp = 0
MatrizPontos[Pallet_2,Prdt_5Aero,2].AbreGarraOp = 0
MatrizPontos[Pallet_2,Prdt_5Aero,2].SensoresCaixa = 12345
MatrizPontos[Pallet_2,Prdt_5Aero,2].TravaGarra = False
MatrizPontos[Pallet_2,Prdt_5Aero,2].SkipGoHome = False
MatrizPontos[Pallet_2,Prdt_5Aero,2].SkipSobeRelAtual = False
MatrizPontos[Pallet_2,Prdt_5Aero,2].XApp1Place=P2_5Aero_2_App1
MatrizPontos[Pallet_2,Prdt_5Aero,2].XApp2Place=P2_5Aero_2_App2
MatrizPontos[Pallet_2,Prdt_5Aero,2].XPlace=P2_5Aero_2_Place
;ENDFOLD
;FOLD OffsetPlace
MatrizPontos[Pallet_2,Prdt_5Aero,2].OffsetPlace.X=0
MatrizPontos[Pallet_2,Prdt_5Aero,2].OffsetPlace.Y=0
MatrizPontos[Pallet_2,Prdt_5Aero,2].OffsetPlace.Z=0
MatrizPontos[Pallet_2,Prdt_5Aero,2].OffsetPlace.A=0
MatrizPontos[Pallet_2,Prdt_5Aero,2].OffsetPlace.B=0
MatrizPontos[Pallet_2,Prdt_5Aero,2].OffsetPlace.C=0
;ENDFOLD
;ENDFOLD

;FOLD PLACE 3
;FOLD PROPRIEDADES
MatrizPontos[Pallet_2,Prdt_5Aero,3].NumCaixas = 3
MatrizPontos[Pallet_2,Prdt_5Aero,3].PickOp = 1
MatrizPontos[Pallet_2,Prdt_5Aero,3].ConfGarraOp = 0
MatrizPontos[Pallet_2,Prdt_5Aero,3].FechaGarraOp = 0
MatrizPontos[Pallet_2,Prdt_5Aero,3].AbreGarraOp = 0
MatrizPontos[Pallet_2,Prdt_5Aero,3].SensoresCaixa = 12345
MatrizPontos[Pallet_2,Prdt_5Aero,3].TravaGarra = False
MatrizPontos[Pallet_2,Prdt_5Aero,3].SkipGoHome = False
MatrizPontos[Pallet_2,Prdt_5Aero,3].SkipSobeRelAtual = False
MatrizPontos[Pallet_2,Prdt_5Aero,3].XApp1Place=P2_5Aero_3_App1
MatrizPontos[Pallet_2,Prdt_5Aero,3].XApp2Place=P2_5Aero_3_App2
MatrizPontos[Pallet_2,Prdt_5Aero,3].XPlace=P2_5Aero_3_Place
;ENDFOLD
;FOLD OffsetPlace
MatrizPontos[Pallet_2,Prdt_5Aero,3].OffsetPlace.X=0
MatrizPontos[Pallet_2,Prdt_5Aero,3].OffsetPlace.Y=0
MatrizPontos[Pallet_2,Prdt_5Aero,3].OffsetPlace.Z=0
MatrizPontos[Pallet_2,Prdt_5Aero,3].OffsetPlace.A=0
MatrizPontos[Pallet_2,Prdt_5Aero,3].OffsetPlace.B=0
MatrizPontos[Pallet_2,Prdt_5Aero,3].OffsetPlace.C=0
;ENDFOLD
;ENDFOLD

;ENDFOLD
;ENDFOLD

;FOLD Pallet 2 - Produto 17KitKat
;FOLD LAYER 1: PLACE 1 ate 4
;FOLD PLACE 1
;FOLD PROPRIEDADES
MatrizPontos[Pallet_2,Prdt_17KitKat,1].NumCaixas = 3
MatrizPontos[Pallet_2,Prdt_17KitKat,1].PickOp = 1
MatrizPontos[Pallet_2,Prdt_17KitKat,1].ConfGarraOp = 0
MatrizPontos[Pallet_2,Prdt_17KitKat,1].FechaGarraOp = 0
MatrizPontos[Pallet_2,Prdt_17KitKat,1].AbreGarraOp = 0
MatrizPontos[Pallet_2,Prdt_17KitKat,1].SensoresCaixa = 1234
MatrizPontos[Pallet_2,Prdt_17KitKat,1].TravaGarra = False
MatrizPontos[Pallet_2,Prdt_17KitKat,1].SkipGoHome = False
MatrizPontos[Pallet_2,Prdt_17KitKat,1].SkipSobeRelAtual = False
MatrizPontos[Pallet_2,Prdt_17KitKat,1].XApp1Place=P2_17KitKat_1_App1
MatrizPontos[Pallet_2,Prdt_17KitKat,1].XApp2Place=P2_17KitKat_1_App2
MatrizPontos[Pallet_2,Prdt_17KitKat,1].XPlace=P2_17KitKat_1_Place
;ENDFOLD
;FOLD OffsetPlace
MatrizPontos[Pallet_2,Prdt_17KitKat,1].OffsetPlace.X=0
MatrizPontos[Pallet_2,Prdt_17KitKat,1].OffsetPlace.Y=0
MatrizPontos[Pallet_2,Prdt_17KitKat,1].OffsetPlace.Z=0
MatrizPontos[Pallet_2,Prdt_17KitKat,1].OffsetPlace.A=0
MatrizPontos[Pallet_2,Prdt_17KitKat,1].OffsetPlace.B=0
MatrizPontos[Pallet_2,Prdt_17KitKat,1].OffsetPlace.C=0
;ENDFOLD
;ENDFOLD

;FOLD PLACE 2
;FOLD PROPRIEDADES
MatrizPontos[Pallet_2,Prdt_17KitKat,2].NumCaixas = 3
MatrizPontos[Pallet_2,Prdt_17KitKat,2].PickOp = 1
MatrizPontos[Pallet_2,Prdt_17KitKat,2].ConfGarraOp = 0
MatrizPontos[Pallet_2,Prdt_17KitKat,2].FechaGarraOp = 0
MatrizPontos[Pallet_2,Prdt_17KitKat,2].AbreGarraOp = 0
MatrizPontos[Pallet_2,Prdt_17KitKat,2].SensoresCaixa = 1234
MatrizPontos[Pallet_2,Prdt_17KitKat,2].TravaGarra = False
MatrizPontos[Pallet_2,Prdt_17KitKat,2].SkipGoHome = False
MatrizPontos[Pallet_2,Prdt_17KitKat,2].SkipSobeRelAtual = False
MatrizPontos[Pallet_2,Prdt_17KitKat,2].XApp1Place=P2_17KitKat_2_App1
MatrizPontos[Pallet_2,Prdt_17KitKat,2].XApp2Place=P2_17KitKat_2_App2
MatrizPontos[Pallet_2,Prdt_17KitKat,2].XPlace=P2_17KitKat_2_Place
;ENDFOLD
;FOLD OffsetPlace
MatrizPontos[Pallet_2,Prdt_17KitKat,2].OffsetPlace.X=0
MatrizPontos[Pallet_2,Prdt_17KitKat,2].OffsetPlace.Y=0
MatrizPontos[Pallet_2,Prdt_17KitKat,2].OffsetPlace.Z=0
MatrizPontos[Pallet_2,Prdt_17KitKat,2].OffsetPlace.A=0
MatrizPontos[Pallet_2,Prdt_17KitKat,2].OffsetPlace.B=0
MatrizPontos[Pallet_2,Prdt_17KitKat,2].OffsetPlace.C=0
;ENDFOLD
;ENDFOLD

;FOLD PLACE 3
;FOLD PROPRIEDADES
MatrizPontos[Pallet_2,Prdt_17KitKat,3].NumCaixas = 3
MatrizPontos[Pallet_2,Prdt_17KitKat,3].PickOp = 1
MatrizPontos[Pallet_2,Prdt_17KitKat,3].ConfGarraOp = 0
MatrizPontos[Pallet_2,Prdt_17KitKat,3].FechaGarraOp = 0
MatrizPontos[Pallet_2,Prdt_17KitKat,3].AbreGarraOp = 0
MatrizPontos[Pallet_2,Prdt_17KitKat,3].SensoresCaixa = 1234
MatrizPontos[Pallet_2,Prdt_17KitKat,3].TravaGarra = False
MatrizPontos[Pallet_2,Prdt_17KitKat,3].SkipGoHome = False
MatrizPontos[Pallet_2,Prdt_17KitKat,3].SkipSobeRelAtual = False
MatrizPontos[Pallet_2,Prdt_17KitKat,3].XApp1Place=P2_17KitKat_3_App1
MatrizPontos[Pallet_2,Prdt_17KitKat,3].XApp2Place=P2_17KitKat_3_App2
MatrizPontos[Pallet_2,Prdt_17KitKat,3].XPlace=P2_17KitKat_3_Place
;ENDFOLD
;FOLD OffsetPlace
MatrizPontos[Pallet_2,Prdt_17KitKat,3].OffsetPlace.X=0
MatrizPontos[Pallet_2,Prdt_17KitKat,3].OffsetPlace.Y=0
MatrizPontos[Pallet_2,Prdt_17KitKat,3].OffsetPlace.Z=0
MatrizPontos[Pallet_2,Prdt_17KitKat,3].OffsetPlace.A=0
MatrizPontos[Pallet_2,Prdt_17KitKat,3].OffsetPlace.B=0
MatrizPontos[Pallet_2,Prdt_17KitKat,3].OffsetPlace.C=0
;ENDFOLD
;ENDFOLD

;FOLD PLACE 4
;FOLD PROPRIEDADES
MatrizPontos[Pallet_2,Prdt_17KitKat,4].NumCaixas = 3
MatrizPontos[Pallet_2,Prdt_17KitKat,4].PickOp = 1
MatrizPontos[Pallet_2,Prdt_17KitKat,4].ConfGarraOp = 0
MatrizPontos[Pallet_2,Prdt_17KitKat,4].FechaGarraOp = 0
MatrizPontos[Pallet_2,Prdt_17KitKat,4].AbreGarraOp = 0
MatrizPontos[Pallet_2,Prdt_17KitKat,4].SensoresCaixa = 1234
MatrizPontos[Pallet_2,Prdt_17KitKat,4].TravaGarra = False
MatrizPontos[Pallet_2,Prdt_17KitKat,4].SkipGoHome = False
MatrizPontos[Pallet_2,Prdt_17KitKat,4].SkipSobeRelAtual = False
MatrizPontos[Pallet_2,Prdt_17KitKat,4].XApp1Place=P2_17KitKat_4_App1
MatrizPontos[Pallet_2,Prdt_17KitKat,4].XApp2Place=P2_17KitKat_4_App2
MatrizPontos[Pallet_2,Prdt_17KitKat,4].XPlace=P2_17KitKat_4_Place
;ENDFOLD
;FOLD OffsetPlace
MatrizPontos[Pallet_2,Prdt_17KitKat,4].OffsetPlace.X=0
MatrizPontos[Pallet_2,Prdt_17KitKat,4].OffsetPlace.Y=0
MatrizPontos[Pallet_2,Prdt_17KitKat,4].OffsetPlace.Z=0
MatrizPontos[Pallet_2,Prdt_17KitKat,4].OffsetPlace.A=0
MatrizPontos[Pallet_2,Prdt_17KitKat,4].OffsetPlace.B=0
MatrizPontos[Pallet_2,Prdt_17KitKat,4].OffsetPlace.C=0
;ENDFOLD
;ENDFOLD

;ENDFOLD
;ENDFOLD

;FOLD Pallet 2 - Produto 20KitKat
;FOLD LAYER 1: PLACE 1 ate 3
;FOLD PLACE 1
;FOLD PROPRIEDADES
MatrizPontos[Pallet_2,Prdt_20KitKat,1].NumCaixas = 4
MatrizPontos[Pallet_2,Prdt_20KitKat,1].PickOp = 1
MatrizPontos[Pallet_2,Prdt_20KitKat,1].ConfGarraOp = 0
MatrizPontos[Pallet_2,Prdt_20KitKat,1].FechaGarraOp = 0
MatrizPontos[Pallet_2,Prdt_20KitKat,1].AbreGarraOp = 0
MatrizPontos[Pallet_2,Prdt_20KitKat,1].SensoresCaixa = 123456
MatrizPontos[Pallet_2,Prdt_20KitKat,1].TravaGarra = False
MatrizPontos[Pallet_2,Prdt_20KitKat,1].SkipGoHome = False
MatrizPontos[Pallet_2,Prdt_20KitKat,1].SkipSobeRelAtual = False
MatrizPontos[Pallet_2,Prdt_20KitKat,1].XApp1Place=P2_20KitKat_1_App1
MatrizPontos[Pallet_2,Prdt_20KitKat,1].XApp2Place=P2_20KitKat_1_App2
MatrizPontos[Pallet_2,Prdt_20KitKat,1].XPlace=P2_20KitKat_1_Place
;ENDFOLD
;FOLD OffsetPlace
MatrizPontos[Pallet_2,Prdt_20KitKat,1].OffsetPlace.X=0
MatrizPontos[Pallet_2,Prdt_20KitKat,1].OffsetPlace.Y=0
MatrizPontos[Pallet_2,Prdt_20KitKat,1].OffsetPlace.Z=0
MatrizPontos[Pallet_2,Prdt_20KitKat,1].OffsetPlace.A=0
MatrizPontos[Pallet_2,Prdt_20KitKat,1].OffsetPlace.B=0
MatrizPontos[Pallet_2,Prdt_20KitKat,1].OffsetPlace.C=0
;ENDFOLD
;ENDFOLD

;FOLD PLACE 2
;FOLD PROPRIEDADES
MatrizPontos[Pallet_2,Prdt_20KitKat,2].NumCaixas = 4
MatrizPontos[Pallet_2,Prdt_20KitKat,2].PickOp = 1
MatrizPontos[Pallet_2,Prdt_20KitKat,2].ConfGarraOp = 0
MatrizPontos[Pallet_2,Prdt_20KitKat,2].FechaGarraOp = 0
MatrizPontos[Pallet_2,Prdt_20KitKat,2].AbreGarraOp = 0
MatrizPontos[Pallet_2,Prdt_20KitKat,2].SensoresCaixa = 123456
MatrizPontos[Pallet_2,Prdt_20KitKat,2].TravaGarra = False
MatrizPontos[Pallet_2,Prdt_20KitKat,2].SkipGoHome = False
MatrizPontos[Pallet_2,Prdt_20KitKat,2].SkipSobeRelAtual = False
MatrizPontos[Pallet_2,Prdt_20KitKat,2].XApp1Place=P2_20KitKat_2_App1
MatrizPontos[Pallet_2,Prdt_20KitKat,2].XApp2Place=P2_20KitKat_2_App2
MatrizPontos[Pallet_2,Prdt_20KitKat,2].XPlace=P2_20KitKat_2_Place
;ENDFOLD
;FOLD OffsetPlace
MatrizPontos[Pallet_2,Prdt_20KitKat,2].OffsetPlace.X=0
MatrizPontos[Pallet_2,Prdt_20KitKat,2].OffsetPlace.Y=0
MatrizPontos[Pallet_2,Prdt_20KitKat,2].OffsetPlace.Z=0
MatrizPontos[Pallet_2,Prdt_20KitKat,2].OffsetPlace.A=0
MatrizPontos[Pallet_2,Prdt_20KitKat,2].OffsetPlace.B=0
MatrizPontos[Pallet_2,Prdt_20KitKat,2].OffsetPlace.C=0
;ENDFOLD
;ENDFOLD

;FOLD PLACE 3
;FOLD PROPRIEDADES
MatrizPontos[Pallet_2,Prdt_20KitKat,3].NumCaixas = 4
MatrizPontos[Pallet_2,Prdt_20KitKat,3].PickOp = 1
MatrizPontos[Pallet_2,Prdt_20KitKat,3].ConfGarraOp = 0
MatrizPontos[Pallet_2,Prdt_20KitKat,3].FechaGarraOp = 0
MatrizPontos[Pallet_2,Prdt_20KitKat,3].AbreGarraOp = 0
MatrizPontos[Pallet_2,Prdt_20KitKat,3].SensoresCaixa = 123456
MatrizPontos[Pallet_2,Prdt_20KitKat,3].TravaGarra = False
MatrizPontos[Pallet_2,Prdt_20KitKat,3].SkipGoHome = False
MatrizPontos[Pallet_2,Prdt_20KitKat,3].SkipSobeRelAtual = False
MatrizPontos[Pallet_2,Prdt_20KitKat,3].XApp1Place=P2_20KitKat_3_App1
MatrizPontos[Pallet_2,Prdt_20KitKat,3].XApp2Place=P2_20KitKat_3_App2
MatrizPontos[Pallet_2,Prdt_20KitKat,3].XPlace=P2_20KitKat_3_Place
;ENDFOLD
;FOLD OffsetPlace
MatrizPontos[Pallet_2,Prdt_20KitKat,3].OffsetPlace.X=0
MatrizPontos[Pallet_2,Prdt_20KitKat,3].OffsetPlace.Y=0
MatrizPontos[Pallet_2,Prdt_20KitKat,3].OffsetPlace.Z=0
MatrizPontos[Pallet_2,Prdt_20KitKat,3].OffsetPlace.A=0
MatrizPontos[Pallet_2,Prdt_20KitKat,3].OffsetPlace.B=0
MatrizPontos[Pallet_2,Prdt_20KitKat,3].OffsetPlace.C=0
;ENDFOLD
;ENDFOLD

;ENDFOLD
;ENDFOLD

;FOLD Pallet 2 - Produto 11CoffeCrisp
;FOLD LAYER 1: PLACE 1 ate 3
;FOLD PLACE 1
;FOLD PROPRIEDADES
MatrizPontos[Pallet_2,Prdt_11CoffeCrisp,1].NumCaixas = 3
MatrizPontos[Pallet_2,Prdt_11CoffeCrisp,1].PickOp = 1
MatrizPontos[Pallet_2,Prdt_11CoffeCrisp,1].ConfGarraOp = 0
MatrizPontos[Pallet_2,Prdt_11CoffeCrisp,1].FechaGarraOp = 0
MatrizPontos[Pallet_2,Prdt_11CoffeCrisp,1].AbreGarraOp = 0
MatrizPontos[Pallet_2,Prdt_11CoffeCrisp,1].SensoresCaixa = 12345
MatrizPontos[Pallet_2,Prdt_11CoffeCrisp,1].TravaGarra = False
MatrizPontos[Pallet_2,Prdt_11CoffeCrisp,1].SkipGoHome = False
MatrizPontos[Pallet_2,Prdt_11CoffeCrisp,1].SkipSobeRelAtual = False
MatrizPontos[Pallet_2,Prdt_11CoffeCrisp,1].XApp1Place=P2_11CoffeCrisp_1_App1
MatrizPontos[Pallet_2,Prdt_11CoffeCrisp,1].XApp2Place=P2_11CoffeCrisp_1_App2
MatrizPontos[Pallet_2,Prdt_11CoffeCrisp,1].XPlace=P2_11CoffeCrisp_1_Place
;ENDFOLD
;FOLD OffsetPlace
MatrizPontos[Pallet_2,Prdt_11CoffeCrisp,1].OffsetPlace.X=0
MatrizPontos[Pallet_2,Prdt_11CoffeCrisp,1].OffsetPlace.Y=0
MatrizPontos[Pallet_2,Prdt_11CoffeCrisp,1].OffsetPlace.Z=0
MatrizPontos[Pallet_2,Prdt_11CoffeCrisp,1].OffsetPlace.A=0
MatrizPontos[Pallet_2,Prdt_11CoffeCrisp,1].OffsetPlace.B=0
MatrizPontos[Pallet_2,Prdt_11CoffeCrisp,1].OffsetPlace.C=0
;ENDFOLD
;ENDFOLD

;FOLD PLACE 2
;FOLD PROPRIEDADES
MatrizPontos[Pallet_2,Prdt_11CoffeCrisp,2].NumCaixas = 3
MatrizPontos[Pallet_2,Prdt_11CoffeCrisp,2].PickOp = 1
MatrizPontos[Pallet_2,Prdt_11CoffeCrisp,2].ConfGarraOp = 0
MatrizPontos[Pallet_2,Prdt_11CoffeCrisp,2].FechaGarraOp = 0
MatrizPontos[Pallet_2,Prdt_11CoffeCrisp,2].AbreGarraOp = 0
MatrizPontos[Pallet_2,Prdt_11CoffeCrisp,2].SensoresCaixa = 12345
MatrizPontos[Pallet_2,Prdt_11CoffeCrisp,2].TravaGarra = False
MatrizPontos[Pallet_2,Prdt_11CoffeCrisp,2].SkipGoHome = False
MatrizPontos[Pallet_2,Prdt_11CoffeCrisp,2].SkipSobeRelAtual = False
MatrizPontos[Pallet_2,Prdt_11CoffeCrisp,2].XApp1Place=P2_11CoffeCrisp_2_App1
MatrizPontos[Pallet_2,Prdt_11CoffeCrisp,2].XApp2Place=P2_11CoffeCrisp_2_App2
MatrizPontos[Pallet_2,Prdt_11CoffeCrisp,2].XPlace=P2_11CoffeCrisp_2_Place
;ENDFOLD
;FOLD OffsetPlace
MatrizPontos[Pallet_2,Prdt_11CoffeCrisp,2].OffsetPlace.X=0
MatrizPontos[Pallet_2,Prdt_11CoffeCrisp,2].OffsetPlace.Y=0
MatrizPontos[Pallet_2,Prdt_11CoffeCrisp,2].OffsetPlace.Z=0
MatrizPontos[Pallet_2,Prdt_11CoffeCrisp,2].OffsetPlace.A=0
MatrizPontos[Pallet_2,Prdt_11CoffeCrisp,2].OffsetPlace.B=0
MatrizPontos[Pallet_2,Prdt_11CoffeCrisp,2].OffsetPlace.C=0
;ENDFOLD
;ENDFOLD

;FOLD PLACE 3
;FOLD PROPRIEDADES
MatrizPontos[Pallet_2,Prdt_11CoffeCrisp,3].NumCaixas = 3
MatrizPontos[Pallet_2,Prdt_11CoffeCrisp,3].PickOp = 1
MatrizPontos[Pallet_2,Prdt_11CoffeCrisp,3].ConfGarraOp = 0
MatrizPontos[Pallet_2,Prdt_11CoffeCrisp,3].FechaGarraOp = 0
MatrizPontos[Pallet_2,Prdt_11CoffeCrisp,3].AbreGarraOp = 0
MatrizPontos[Pallet_2,Prdt_11CoffeCrisp,3].SensoresCaixa = 12345
MatrizPontos[Pallet_2,Prdt_11CoffeCrisp,3].TravaGarra = False
MatrizPontos[Pallet_2,Prdt_11CoffeCrisp,3].SkipGoHome = False
MatrizPontos[Pallet_2,Prdt_11CoffeCrisp,3].SkipSobeRelAtual = False
MatrizPontos[Pallet_2,Prdt_11CoffeCrisp,3].XApp1Place=P2_11CoffeCrisp_3_App1
MatrizPontos[Pallet_2,Prdt_11CoffeCrisp,3].XApp2Place=P2_11CoffeCrisp_3_App2
MatrizPontos[Pallet_2,Prdt_11CoffeCrisp,3].XPlace=P2_11CoffeCrisp_3_Place
;ENDFOLD
;FOLD OffsetPlace
MatrizPontos[Pallet_2,Prdt_11CoffeCrisp,3].OffsetPlace.X=0
MatrizPontos[Pallet_2,Prdt_11CoffeCrisp,3].OffsetPlace.Y=0
MatrizPontos[Pallet_2,Prdt_11CoffeCrisp,3].OffsetPlace.Z=0
MatrizPontos[Pallet_2,Prdt_11CoffeCrisp,3].OffsetPlace.A=0
MatrizPontos[Pallet_2,Prdt_11CoffeCrisp,3].OffsetPlace.B=0
MatrizPontos[Pallet_2,Prdt_11CoffeCrisp,3].OffsetPlace.C=0
;ENDFOLD
;ENDFOLD

;ENDFOLD
;ENDFOLD

;FOLD Pallet 2 - Produto 21KitKat
;FOLD LAYER 1: PLACE 1 ate 3
;FOLD PLACE 1
;FOLD PROPRIEDADES
MatrizPontos[Pallet_2,Prdt_21KitKat,1].NumCaixas = 4
MatrizPontos[Pallet_2,Prdt_21KitKat,1].PickOp = 1
MatrizPontos[Pallet_2,Prdt_21KitKat,1].ConfGarraOp = 0
MatrizPontos[Pallet_2,Prdt_21KitKat,1].FechaGarraOp = 0
MatrizPontos[Pallet_2,Prdt_21KitKat,1].AbreGarraOp = 0
MatrizPontos[Pallet_2,Prdt_21KitKat,1].SensoresCaixa = 12345
MatrizPontos[Pallet_2,Prdt_21KitKat,1].TravaGarra = False
MatrizPontos[Pallet_2,Prdt_21KitKat,1].SkipGoHome = False
MatrizPontos[Pallet_2,Prdt_21KitKat,1].SkipSobeRelAtual = False
MatrizPontos[Pallet_2,Prdt_21KitKat,1].XApp1Place=P2_21KitKat_1_App1
MatrizPontos[Pallet_2,Prdt_21KitKat,1].XApp2Place=P2_21KitKat_1_App2
MatrizPontos[Pallet_2,Prdt_21KitKat,1].XPlace=P2_21KitKat_1_Place
;ENDFOLD
;FOLD OffsetPlace
MatrizPontos[Pallet_2,Prdt_21KitKat,1].OffsetPlace.X=0
MatrizPontos[Pallet_2,Prdt_21KitKat,1].OffsetPlace.Y=0
MatrizPontos[Pallet_2,Prdt_21KitKat,1].OffsetPlace.Z=0
MatrizPontos[Pallet_2,Prdt_21KitKat,1].OffsetPlace.A=0
MatrizPontos[Pallet_2,Prdt_21KitKat,1].OffsetPlace.B=0
MatrizPontos[Pallet_2,Prdt_21KitKat,1].OffsetPlace.C=0
;ENDFOLD
;ENDFOLD

;FOLD PLACE 2
;FOLD PROPRIEDADES
MatrizPontos[Pallet_2,Prdt_21KitKat,2].NumCaixas = 4
MatrizPontos[Pallet_2,Prdt_21KitKat,2].PickOp = 1
MatrizPontos[Pallet_2,Prdt_21KitKat,2].ConfGarraOp = 0
MatrizPontos[Pallet_2,Prdt_21KitKat,2].FechaGarraOp = 0
MatrizPontos[Pallet_2,Prdt_21KitKat,2].AbreGarraOp = 0
MatrizPontos[Pallet_2,Prdt_21KitKat,2].SensoresCaixa = 12345
MatrizPontos[Pallet_2,Prdt_21KitKat,2].TravaGarra = False
MatrizPontos[Pallet_2,Prdt_21KitKat,2].SkipGoHome = False
MatrizPontos[Pallet_2,Prdt_21KitKat,2].SkipSobeRelAtual = False
MatrizPontos[Pallet_2,Prdt_21KitKat,2].XApp1Place=P2_21KitKat_2_App1
MatrizPontos[Pallet_2,Prdt_21KitKat,2].XApp2Place=P2_21KitKat_2_App2
MatrizPontos[Pallet_2,Prdt_21KitKat,2].XPlace=P2_21KitKat_2_Place
;ENDFOLD
;FOLD OffsetPlace
MatrizPontos[Pallet_2,Prdt_21KitKat,2].OffsetPlace.X=0
MatrizPontos[Pallet_2,Prdt_21KitKat,2].OffsetPlace.Y=0
MatrizPontos[Pallet_2,Prdt_21KitKat,2].OffsetPlace.Z=0
MatrizPontos[Pallet_2,Prdt_21KitKat,2].OffsetPlace.A=0
MatrizPontos[Pallet_2,Prdt_21KitKat,2].OffsetPlace.B=0
MatrizPontos[Pallet_2,Prdt_21KitKat,2].OffsetPlace.C=0
;ENDFOLD
;ENDFOLD

;FOLD PLACE 3
;FOLD PROPRIEDADES
MatrizPontos[Pallet_2,Prdt_21KitKat,3].NumCaixas = 4
MatrizPontos[Pallet_2,Prdt_21KitKat,3].PickOp = 1
MatrizPontos[Pallet_2,Prdt_21KitKat,3].ConfGarraOp = 0
MatrizPontos[Pallet_2,Prdt_21KitKat,3].FechaGarraOp = 0
MatrizPontos[Pallet_2,Prdt_21KitKat,3].AbreGarraOp = 0
MatrizPontos[Pallet_2,Prdt_21KitKat,3].SensoresCaixa = 12345
MatrizPontos[Pallet_2,Prdt_21KitKat,3].TravaGarra = False
MatrizPontos[Pallet_2,Prdt_21KitKat,3].SkipGoHome = False
MatrizPontos[Pallet_2,Prdt_21KitKat,3].SkipSobeRelAtual = False
MatrizPontos[Pallet_2,Prdt_21KitKat,3].XApp1Place=P2_21KitKat_3_App1
MatrizPontos[Pallet_2,Prdt_21KitKat,3].XApp2Place=P2_21KitKat_3_App2
MatrizPontos[Pallet_2,Prdt_21KitKat,3].XPlace=P2_21KitKat_3_Place
;ENDFOLD
;FOLD OffsetPlace
MatrizPontos[Pallet_2,Prdt_21KitKat,3].OffsetPlace.X=0
MatrizPontos[Pallet_2,Prdt_21KitKat,3].OffsetPlace.Y=0
MatrizPontos[Pallet_2,Prdt_21KitKat,3].OffsetPlace.Z=0
MatrizPontos[Pallet_2,Prdt_21KitKat,3].OffsetPlace.A=0
MatrizPontos[Pallet_2,Prdt_21KitKat,3].OffsetPlace.B=0
MatrizPontos[Pallet_2,Prdt_21KitKat,3].OffsetPlace.C=0
;ENDFOLD
;ENDFOLD

;ENDFOLD
;ENDFOLD

;FOLD Pallet 2 - Produto 30All
;FOLD LAYER 1: PLACE 1 ate 4
;FOLD PLACE 1
;FOLD PROPRIEDADES
MatrizPontos[Pallet_2,Prdt_30All,1].NumCaixas = 4
MatrizPontos[Pallet_2,Prdt_30All,1].PickOp = 1
MatrizPontos[Pallet_2,Prdt_30All,1].ConfGarraOp = 0
MatrizPontos[Pallet_2,Prdt_30All,1].FechaGarraOp = 0
MatrizPontos[Pallet_2,Prdt_30All,1].AbreGarraOp = 0
MatrizPontos[Pallet_2,Prdt_30All,1].SensoresCaixa = 12345
MatrizPontos[Pallet_2,Prdt_30All,1].TravaGarra = False
MatrizPontos[Pallet_2,Prdt_30All,1].SkipGoHome = False
MatrizPontos[Pallet_2,Prdt_30All,1].SkipSobeRelAtual = False
MatrizPontos[Pallet_2,Prdt_30All,1].XApp1Place=P2_30All_1_App1
MatrizPontos[Pallet_2,Prdt_30All,1].XApp2Place=P2_30All_1_App2
MatrizPontos[Pallet_2,Prdt_30All,1].XPlace=P2_30All_1_Place
;ENDFOLD
;FOLD OffsetPlace
MatrizPontos[Pallet_2,Prdt_30All,1].OffsetPlace.X=0
MatrizPontos[Pallet_2,Prdt_30All,1].OffsetPlace.Y=0
MatrizPontos[Pallet_2,Prdt_30All,1].OffsetPlace.Z=0
MatrizPontos[Pallet_2,Prdt_30All,1].OffsetPlace.A=0
MatrizPontos[Pallet_2,Prdt_30All,1].OffsetPlace.B=0
MatrizPontos[Pallet_2,Prdt_30All,1].OffsetPlace.C=0
;ENDFOLD
;ENDFOLD

;FOLD PLACE 2
;FOLD PROPRIEDADES
MatrizPontos[Pallet_2,Prdt_30All,2].NumCaixas = 4
MatrizPontos[Pallet_2,Prdt_30All,2].PickOp = 1
MatrizPontos[Pallet_2,Prdt_30All,2].ConfGarraOp = 0
MatrizPontos[Pallet_2,Prdt_30All,2].FechaGarraOp = 0
MatrizPontos[Pallet_2,Prdt_30All,2].AbreGarraOp = 0
MatrizPontos[Pallet_2,Prdt_30All,2].SensoresCaixa = 12345
MatrizPontos[Pallet_2,Prdt_30All,2].TravaGarra = False
MatrizPontos[Pallet_2,Prdt_30All,2].SkipGoHome = False
MatrizPontos[Pallet_2,Prdt_30All,2].SkipSobeRelAtual = False
MatrizPontos[Pallet_2,Prdt_30All,2].XApp1Place=P2_30All_2_App1
MatrizPontos[Pallet_2,Prdt_30All,2].XApp2Place=P2_30All_2_App2
MatrizPontos[Pallet_2,Prdt_30All,2].XPlace=P2_30All_2_Place
;ENDFOLD
;FOLD OffsetPlace
MatrizPontos[Pallet_2,Prdt_30All,2].OffsetPlace.X=0
MatrizPontos[Pallet_2,Prdt_30All,2].OffsetPlace.Y=0
MatrizPontos[Pallet_2,Prdt_30All,2].OffsetPlace.Z=0
MatrizPontos[Pallet_2,Prdt_30All,2].OffsetPlace.A=0
MatrizPontos[Pallet_2,Prdt_30All,2].OffsetPlace.B=0
MatrizPontos[Pallet_2,Prdt_30All,2].OffsetPlace.C=0
;ENDFOLD
;ENDFOLD

;FOLD PLACE 3
;FOLD PROPRIEDADES
MatrizPontos[Pallet_2,Prdt_30All,3].NumCaixas = 4
MatrizPontos[Pallet_2,Prdt_30All,3].PickOp = 1
MatrizPontos[Pallet_2,Prdt_30All,3].ConfGarraOp = 0
MatrizPontos[Pallet_2,Prdt_30All,3].FechaGarraOp = 0
MatrizPontos[Pallet_2,Prdt_30All,3].AbreGarraOp = 0
MatrizPontos[Pallet_2,Prdt_30All,3].SensoresCaixa = 12345
MatrizPontos[Pallet_2,Prdt_30All,3].TravaGarra = False
MatrizPontos[Pallet_2,Prdt_30All,3].SkipGoHome = False
MatrizPontos[Pallet_2,Prdt_30All,3].SkipSobeRelAtual = False
MatrizPontos[Pallet_2,Prdt_30All,3].XApp1Place=P2_30All_3_App1
MatrizPontos[Pallet_2,Prdt_30All,3].XApp2Place=P2_30All_3_App2
MatrizPontos[Pallet_2,Prdt_30All,3].XPlace=P2_30All_3_Place
;ENDFOLD
;FOLD OffsetPlace
MatrizPontos[Pallet_2,Prdt_30All,3].OffsetPlace.X=0
MatrizPontos[Pallet_2,Prdt_30All,3].OffsetPlace.Y=0
MatrizPontos[Pallet_2,Prdt_30All,3].OffsetPlace.Z=0
MatrizPontos[Pallet_2,Prdt_30All,3].OffsetPlace.A=0
MatrizPontos[Pallet_2,Prdt_30All,3].OffsetPlace.B=0
MatrizPontos[Pallet_2,Prdt_30All,3].OffsetPlace.C=0
;ENDFOLD
;ENDFOLD

;FOLD PLACE 4
;FOLD PROPRIEDADES
MatrizPontos[Pallet_2,Prdt_30All,4].NumCaixas = 4
MatrizPontos[Pallet_2,Prdt_30All,4].PickOp = 1
MatrizPontos[Pallet_2,Prdt_30All,4].ConfGarraOp = 0
MatrizPontos[Pallet_2,Prdt_30All,4].FechaGarraOp = 0
MatrizPontos[Pallet_2,Prdt_30All,4].AbreGarraOp = 0
MatrizPontos[Pallet_2,Prdt_30All,4].SensoresCaixa = 12345
MatrizPontos[Pallet_2,Prdt_30All,4].TravaGarra = False
MatrizPontos[Pallet_2,Prdt_30All,4].SkipGoHome = False
MatrizPontos[Pallet_2,Prdt_30All,4].SkipSobeRelAtual = False
MatrizPontos[Pallet_2,Prdt_30All,4].XApp1Place=P2_30All_4_App1
MatrizPontos[Pallet_2,Prdt_30All,4].XApp2Place=P2_30All_4_App2
MatrizPontos[Pallet_2,Prdt_30All,4].XPlace=P2_30All_4_Place
;ENDFOLD
;FOLD OffsetPlace
MatrizPontos[Pallet_2,Prdt_30All,4].OffsetPlace.X=0
MatrizPontos[Pallet_2,Prdt_30All,4].OffsetPlace.Y=0
MatrizPontos[Pallet_2,Prdt_30All,4].OffsetPlace.Z=0
MatrizPontos[Pallet_2,Prdt_30All,4].OffsetPlace.A=0
MatrizPontos[Pallet_2,Prdt_30All,4].OffsetPlace.B=0
MatrizPontos[Pallet_2,Prdt_30All,4].OffsetPlace.C=0
;ENDFOLD
;ENDFOLD

;ENDFOLD
;ENDFOLD

;FOLD Pallet 2 - Produto 24a28All
;FOLD LAYER 1: PLACE 1 ate 3
;FOLD PLACE 1
;FOLD PROPRIEDADES
MatrizPontos[Pallet_2,Prdt_24a28All,1].NumCaixas = 5
MatrizPontos[Pallet_2,Prdt_24a28All,1].PickOp = 1
MatrizPontos[Pallet_2,Prdt_24a28All,1].ConfGarraOp = 0
MatrizPontos[Pallet_2,Prdt_24a28All,1].FechaGarraOp = 0
MatrizPontos[Pallet_2,Prdt_24a28All,1].AbreGarraOp = 0
MatrizPontos[Pallet_2,Prdt_24a28All,1].SensoresCaixa = 123456
MatrizPontos[Pallet_2,Prdt_24a28All,1].TravaGarra = False
MatrizPontos[Pallet_2,Prdt_24a28All,1].SkipGoHome = False
MatrizPontos[Pallet_2,Prdt_24a28All,1].SkipSobeRelAtual = False
MatrizPontos[Pallet_2,Prdt_24a28All,1].XApp1Place=P2_24a28All_1_App1
MatrizPontos[Pallet_2,Prdt_24a28All,1].XApp2Place=P2_24a28All_1_App2
MatrizPontos[Pallet_2,Prdt_24a28All,1].XPlace=P2_24a28All_1_Place
;ENDFOLD
;FOLD OffsetPlace
MatrizPontos[Pallet_2,Prdt_24a28All,1].OffsetPlace.X=0
MatrizPontos[Pallet_2,Prdt_24a28All,1].OffsetPlace.Y=0
MatrizPontos[Pallet_2,Prdt_24a28All,1].OffsetPlace.Z=0
MatrizPontos[Pallet_2,Prdt_24a28All,1].OffsetPlace.A=0
MatrizPontos[Pallet_2,Prdt_24a28All,1].OffsetPlace.B=0
MatrizPontos[Pallet_2,Prdt_24a28All,1].OffsetPlace.C=0
;ENDFOLD
;ENDFOLD

;FOLD PLACE 2
;FOLD PROPRIEDADES
MatrizPontos[Pallet_2,Prdt_24a28All,2].NumCaixas = 5
MatrizPontos[Pallet_2,Prdt_24a28All,2].PickOp = 1
MatrizPontos[Pallet_2,Prdt_24a28All,2].ConfGarraOp = 0
MatrizPontos[Pallet_2,Prdt_24a28All,2].FechaGarraOp = 0
MatrizPontos[Pallet_2,Prdt_24a28All,2].AbreGarraOp = 0
MatrizPontos[Pallet_2,Prdt_24a28All,2].SensoresCaixa = 123456
MatrizPontos[Pallet_2,Prdt_24a28All,2].TravaGarra = False
MatrizPontos[Pallet_2,Prdt_24a28All,2].SkipGoHome = False
MatrizPontos[Pallet_2,Prdt_24a28All,2].SkipSobeRelAtual = False
MatrizPontos[Pallet_2,Prdt_24a28All,2].XApp1Place=P2_24a28All_2_App1
MatrizPontos[Pallet_2,Prdt_24a28All,2].XApp2Place=P2_24a28All_2_App2
MatrizPontos[Pallet_2,Prdt_24a28All,2].XPlace=P2_24a28All_2_Place
;ENDFOLD
;FOLD OffsetPlace
MatrizPontos[Pallet_2,Prdt_24a28All,2].OffsetPlace.X=0
MatrizPontos[Pallet_2,Prdt_24a28All,2].OffsetPlace.Y=0
MatrizPontos[Pallet_2,Prdt_24a28All,2].OffsetPlace.Z=0
MatrizPontos[Pallet_2,Prdt_24a28All,2].OffsetPlace.A=0
MatrizPontos[Pallet_2,Prdt_24a28All,2].OffsetPlace.B=0
MatrizPontos[Pallet_2,Prdt_24a28All,2].OffsetPlace.C=0
;ENDFOLD
;ENDFOLD

;FOLD PLACE 3
;FOLD PROPRIEDADES
MatrizPontos[Pallet_2,Prdt_24a28All,3].NumCaixas = 5
MatrizPontos[Pallet_2,Prdt_24a28All,3].PickOp = 1
MatrizPontos[Pallet_2,Prdt_24a28All,3].ConfGarraOp = 0
MatrizPontos[Pallet_2,Prdt_24a28All,3].FechaGarraOp = 0
MatrizPontos[Pallet_2,Prdt_24a28All,3].AbreGarraOp = 0
MatrizPontos[Pallet_2,Prdt_24a28All,3].SensoresCaixa = 123456
MatrizPontos[Pallet_2,Prdt_24a28All,3].TravaGarra = False
MatrizPontos[Pallet_2,Prdt_24a28All,3].SkipGoHome = False
MatrizPontos[Pallet_2,Prdt_24a28All,3].SkipSobeRelAtual = False
MatrizPontos[Pallet_2,Prdt_24a28All,3].XApp1Place=P2_24a28All_3_App1
MatrizPontos[Pallet_2,Prdt_24a28All,3].XApp2Place=P2_24a28All_3_App2
MatrizPontos[Pallet_2,Prdt_24a28All,3].XPlace=P2_24a28All_3_Place
;ENDFOLD
;FOLD OffsetPlace
MatrizPontos[Pallet_2,Prdt_24a28All,3].OffsetPlace.X=0
MatrizPontos[Pallet_2,Prdt_24a28All,3].OffsetPlace.Y=0
MatrizPontos[Pallet_2,Prdt_24a28All,3].OffsetPlace.Z=0
MatrizPontos[Pallet_2,Prdt_24a28All,3].OffsetPlace.A=0
MatrizPontos[Pallet_2,Prdt_24a28All,3].OffsetPlace.B=0
MatrizPontos[Pallet_2,Prdt_24a28All,3].OffsetPlace.C=0
;ENDFOLD
;ENDFOLD

;ENDFOLD
;ENDFOLD

;FOLD Pallet 2 - Produto 16CoffeCrisp
;FOLD LAYER 1: PLACE 1 ate 4
;FOLD PLACE 1
;FOLD PROPRIEDADES
MatrizPontos[Pallet_2,Prdt_16CoffeCrisp,1].NumCaixas = 2
MatrizPontos[Pallet_2,Prdt_16CoffeCrisp,1].PickOp = 1
MatrizPontos[Pallet_2,Prdt_16CoffeCrisp,1].ConfGarraOp = 0
MatrizPontos[Pallet_2,Prdt_16CoffeCrisp,1].FechaGarraOp = 0
MatrizPontos[Pallet_2,Prdt_16CoffeCrisp,1].AbreGarraOp = 0
MatrizPontos[Pallet_2,Prdt_16CoffeCrisp,1].SensoresCaixa = 123
MatrizPontos[Pallet_2,Prdt_16CoffeCrisp,1].TravaGarra = False
MatrizPontos[Pallet_2,Prdt_16CoffeCrisp,1].SkipGoHome = False
MatrizPontos[Pallet_2,Prdt_16CoffeCrisp,1].SkipSobeRelAtual = False
MatrizPontos[Pallet_2,Prdt_16CoffeCrisp,1].XApp1Place=P2_16CoffeCrisp_1_App1
MatrizPontos[Pallet_2,Prdt_16CoffeCrisp,1].XApp2Place=P2_16CoffeCrisp_1_App2
MatrizPontos[Pallet_2,Prdt_16CoffeCrisp,1].XPlace=P2_16CoffeCrisp_1_Place
;ENDFOLD
;FOLD OffsetPlace
MatrizPontos[Pallet_2,Prdt_16CoffeCrisp,1].OffsetPlace.X=0
MatrizPontos[Pallet_2,Prdt_16CoffeCrisp,1].OffsetPlace.Y=0
MatrizPontos[Pallet_2,Prdt_16CoffeCrisp,1].OffsetPlace.Z=0
MatrizPontos[Pallet_2,Prdt_16CoffeCrisp,1].OffsetPlace.A=0
MatrizPontos[Pallet_2,Prdt_16CoffeCrisp,1].OffsetPlace.B=0
MatrizPontos[Pallet_2,Prdt_16CoffeCrisp,1].OffsetPlace.C=0
;ENDFOLD
;ENDFOLD

;FOLD PLACE 2
;FOLD PROPRIEDADES
MatrizPontos[Pallet_2,Prdt_16CoffeCrisp,2].NumCaixas = 2
MatrizPontos[Pallet_2,Prdt_16CoffeCrisp,2].PickOp = 1
MatrizPontos[Pallet_2,Prdt_16CoffeCrisp,2].ConfGarraOp = 0
MatrizPontos[Pallet_2,Prdt_16CoffeCrisp,2].FechaGarraOp = 0
MatrizPontos[Pallet_2,Prdt_16CoffeCrisp,2].AbreGarraOp = 0
MatrizPontos[Pallet_2,Prdt_16CoffeCrisp,2].SensoresCaixa = 123
MatrizPontos[Pallet_2,Prdt_16CoffeCrisp,2].TravaGarra = False
MatrizPontos[Pallet_2,Prdt_16CoffeCrisp,2].SkipGoHome = False
MatrizPontos[Pallet_2,Prdt_16CoffeCrisp,2].SkipSobeRelAtual = False
MatrizPontos[Pallet_2,Prdt_16CoffeCrisp,2].XApp1Place=P2_16CoffeCrisp_2_App1
MatrizPontos[Pallet_2,Prdt_16CoffeCrisp,2].XApp2Place=P2_16CoffeCrisp_2_App2
MatrizPontos[Pallet_2,Prdt_16CoffeCrisp,2].XPlace=P2_16CoffeCrisp_2_Place
;ENDFOLD
;FOLD OffsetPlace
MatrizPontos[Pallet_2,Prdt_16CoffeCrisp,2].OffsetPlace.X=0
MatrizPontos[Pallet_2,Prdt_16CoffeCrisp,2].OffsetPlace.Y=0
MatrizPontos[Pallet_2,Prdt_16CoffeCrisp,2].OffsetPlace.Z=0
MatrizPontos[Pallet_2,Prdt_16CoffeCrisp,2].OffsetPlace.A=0
MatrizPontos[Pallet_2,Prdt_16CoffeCrisp,2].OffsetPlace.B=0
MatrizPontos[Pallet_2,Prdt_16CoffeCrisp,2].OffsetPlace.C=0
;ENDFOLD
;ENDFOLD

;FOLD PLACE 3
;FOLD PROPRIEDADES
MatrizPontos[Pallet_2,Prdt_16CoffeCrisp,3].NumCaixas = 2
MatrizPontos[Pallet_2,Prdt_16CoffeCrisp,3].PickOp = 1
MatrizPontos[Pallet_2,Prdt_16CoffeCrisp,3].ConfGarraOp = 0
MatrizPontos[Pallet_2,Prdt_16CoffeCrisp,3].FechaGarraOp = 0
MatrizPontos[Pallet_2,Prdt_16CoffeCrisp,3].AbreGarraOp = 0
MatrizPontos[Pallet_2,Prdt_16CoffeCrisp,3].SensoresCaixa = 123
MatrizPontos[Pallet_2,Prdt_16CoffeCrisp,3].TravaGarra = False
MatrizPontos[Pallet_2,Prdt_16CoffeCrisp,3].SkipGoHome = False
MatrizPontos[Pallet_2,Prdt_16CoffeCrisp,3].SkipSobeRelAtual = False
MatrizPontos[Pallet_2,Prdt_16CoffeCrisp,3].XApp1Place=P2_16CoffeCrisp_3_App1
MatrizPontos[Pallet_2,Prdt_16CoffeCrisp,3].XApp2Place=P2_16CoffeCrisp_3_App2
MatrizPontos[Pallet_2,Prdt_16CoffeCrisp,3].XPlace=P2_16CoffeCrisp_3_Place
;ENDFOLD
;FOLD OffsetPlace
MatrizPontos[Pallet_2,Prdt_16CoffeCrisp,3].OffsetPlace.X=0
MatrizPontos[Pallet_2,Prdt_16CoffeCrisp,3].OffsetPlace.Y=0
MatrizPontos[Pallet_2,Prdt_16CoffeCrisp,3].OffsetPlace.Z=0
MatrizPontos[Pallet_2,Prdt_16CoffeCrisp,3].OffsetPlace.A=0
MatrizPontos[Pallet_2,Prdt_16CoffeCrisp,3].OffsetPlace.B=0
MatrizPontos[Pallet_2,Prdt_16CoffeCrisp,3].OffsetPlace.C=0
;ENDFOLD
;ENDFOLD

;FOLD PLACE 4
;FOLD PROPRIEDADES
MatrizPontos[Pallet_2,Prdt_16CoffeCrisp,4].NumCaixas = 4
MatrizPontos[Pallet_2,Prdt_16CoffeCrisp,4].PickOp = 1
MatrizPontos[Pallet_2,Prdt_16CoffeCrisp,4].ConfGarraOp = 0
MatrizPontos[Pallet_2,Prdt_16CoffeCrisp,4].FechaGarraOp = 0
MatrizPontos[Pallet_2,Prdt_16CoffeCrisp,4].AbreGarraOp = 0
MatrizPontos[Pallet_2,Prdt_16CoffeCrisp,4].SensoresCaixa = 123456
MatrizPontos[Pallet_2,Prdt_16CoffeCrisp,4].TravaGarra = False
MatrizPontos[Pallet_2,Prdt_16CoffeCrisp,4].SkipGoHome = False
MatrizPontos[Pallet_2,Prdt_16CoffeCrisp,4].SkipSobeRelAtual = False
MatrizPontos[Pallet_2,Prdt_16CoffeCrisp,4].XApp1Place=P2_16CoffeCrisp_4_App1
MatrizPontos[Pallet_2,Prdt_16CoffeCrisp,4].XApp2Place=P2_16CoffeCrisp_4_App2
MatrizPontos[Pallet_2,Prdt_16CoffeCrisp,4].XPlace=P2_16CoffeCrisp_4_Place
;ENDFOLD
;FOLD OffsetPlace
MatrizPontos[Pallet_2,Prdt_16CoffeCrisp,4].OffsetPlace.X=0
MatrizPontos[Pallet_2,Prdt_16CoffeCrisp,4].OffsetPlace.Y=0
MatrizPontos[Pallet_2,Prdt_16CoffeCrisp,4].OffsetPlace.Z=0
MatrizPontos[Pallet_2,Prdt_16CoffeCrisp,4].OffsetPlace.A=0
MatrizPontos[Pallet_2,Prdt_16CoffeCrisp,4].OffsetPlace.B=0
MatrizPontos[Pallet_2,Prdt_16CoffeCrisp,4].OffsetPlace.C=0
;ENDFOLD
;ENDFOLD

;ENDFOLD
;FOLD LAYER 2: PLACE 5 ate 8
;FOLD PLACE 5
;FOLD PROPRIEDADES
MatrizPontos[Pallet_2,Prdt_16CoffeCrisp,5].NumCaixas = 4
MatrizPontos[Pallet_2,Prdt_16CoffeCrisp,5].PickOp = 1
MatrizPontos[Pallet_2,Prdt_16CoffeCrisp,5].ConfGarraOp = 0
MatrizPontos[Pallet_2,Prdt_16CoffeCrisp,5].FechaGarraOp = 0
MatrizPontos[Pallet_2,Prdt_16CoffeCrisp,5].AbreGarraOp = 0
MatrizPontos[Pallet_2,Prdt_16CoffeCrisp,5].SensoresCaixa = 123456
MatrizPontos[Pallet_2,Prdt_16CoffeCrisp,5].TravaGarra = False
MatrizPontos[Pallet_2,Prdt_16CoffeCrisp,5].SkipGoHome = False
MatrizPontos[Pallet_2,Prdt_16CoffeCrisp,5].SkipSobeRelAtual = False
MatrizPontos[Pallet_2,Prdt_16CoffeCrisp,5].XApp1Place=P2_16CoffeCrisp_5_App1
MatrizPontos[Pallet_2,Prdt_16CoffeCrisp,5].XApp2Place=P2_16CoffeCrisp_5_App2
MatrizPontos[Pallet_2,Prdt_16CoffeCrisp,5].XPlace=P2_16CoffeCrisp_5_Place
;ENDFOLD
;FOLD OffsetPlace
MatrizPontos[Pallet_2,Prdt_16CoffeCrisp,5].OffsetPlace.X=0
MatrizPontos[Pallet_2,Prdt_16CoffeCrisp,5].OffsetPlace.Y=0
MatrizPontos[Pallet_2,Prdt_16CoffeCrisp,5].OffsetPlace.Z=0
MatrizPontos[Pallet_2,Prdt_16CoffeCrisp,5].OffsetPlace.A=0
MatrizPontos[Pallet_2,Prdt_16CoffeCrisp,5].OffsetPlace.B=0
MatrizPontos[Pallet_2,Prdt_16CoffeCrisp,5].OffsetPlace.C=0
;ENDFOLD
;ENDFOLD

;FOLD PLACE 6
;FOLD PROPRIEDADES
MatrizPontos[Pallet_2,Prdt_16CoffeCrisp,6].NumCaixas = 2
MatrizPontos[Pallet_2,Prdt_16CoffeCrisp,6].PickOp = 1
MatrizPontos[Pallet_2,Prdt_16CoffeCrisp,6].ConfGarraOp = 0
MatrizPontos[Pallet_2,Prdt_16CoffeCrisp,6].FechaGarraOp = 0
MatrizPontos[Pallet_2,Prdt_16CoffeCrisp,6].AbreGarraOp = 0
MatrizPontos[Pallet_2,Prdt_16CoffeCrisp,6].SensoresCaixa = 123
MatrizPontos[Pallet_2,Prdt_16CoffeCrisp,6].TravaGarra = False
MatrizPontos[Pallet_2,Prdt_16CoffeCrisp,6].SkipGoHome = False
MatrizPontos[Pallet_2,Prdt_16CoffeCrisp,6].SkipSobeRelAtual = False
MatrizPontos[Pallet_2,Prdt_16CoffeCrisp,6].XApp1Place=P2_16CoffeCrisp_6_App1
MatrizPontos[Pallet_2,Prdt_16CoffeCrisp,6].XApp2Place=P2_16CoffeCrisp_6_App2
MatrizPontos[Pallet_2,Prdt_16CoffeCrisp,6].XPlace=P2_16CoffeCrisp_6_Place
;ENDFOLD
;FOLD OffsetPlace
MatrizPontos[Pallet_2,Prdt_16CoffeCrisp,6].OffsetPlace.X=0
MatrizPontos[Pallet_2,Prdt_16CoffeCrisp,6].OffsetPlace.Y=0
MatrizPontos[Pallet_2,Prdt_16CoffeCrisp,6].OffsetPlace.Z=0
MatrizPontos[Pallet_2,Prdt_16CoffeCrisp,6].OffsetPlace.A=0
MatrizPontos[Pallet_2,Prdt_16CoffeCrisp,6].OffsetPlace.B=0
MatrizPontos[Pallet_2,Prdt_16CoffeCrisp,6].OffsetPlace.C=0
;ENDFOLD
;ENDFOLD

;FOLD PLACE 7
;FOLD PROPRIEDADES
MatrizPontos[Pallet_2,Prdt_16CoffeCrisp,7].NumCaixas = 2
MatrizPontos[Pallet_2,Prdt_16CoffeCrisp,7].PickOp = 1
MatrizPontos[Pallet_2,Prdt_16CoffeCrisp,7].ConfGarraOp = 0
MatrizPontos[Pallet_2,Prdt_16CoffeCrisp,7].FechaGarraOp = 0
MatrizPontos[Pallet_2,Prdt_16CoffeCrisp,7].AbreGarraOp = 0
MatrizPontos[Pallet_2,Prdt_16CoffeCrisp,7].SensoresCaixa = 123
MatrizPontos[Pallet_2,Prdt_16CoffeCrisp,7].TravaGarra = False
MatrizPontos[Pallet_2,Prdt_16CoffeCrisp,7].SkipGoHome = False
MatrizPontos[Pallet_2,Prdt_16CoffeCrisp,7].SkipSobeRelAtual = False
MatrizPontos[Pallet_2,Prdt_16CoffeCrisp,7].XApp1Place=P2_16CoffeCrisp_7_App1
MatrizPontos[Pallet_2,Prdt_16CoffeCrisp,7].XApp2Place=P2_16CoffeCrisp_7_App2
MatrizPontos[Pallet_2,Prdt_16CoffeCrisp,7].XPlace=P2_16CoffeCrisp_7_Place
;ENDFOLD
;FOLD OffsetPlace
MatrizPontos[Pallet_2,Prdt_16CoffeCrisp,7].OffsetPlace.X=0
MatrizPontos[Pallet_2,Prdt_16CoffeCrisp,7].OffsetPlace.Y=0
MatrizPontos[Pallet_2,Prdt_16CoffeCrisp,7].OffsetPlace.Z=0
MatrizPontos[Pallet_2,Prdt_16CoffeCrisp,7].OffsetPlace.A=0
MatrizPontos[Pallet_2,Prdt_16CoffeCrisp,7].OffsetPlace.B=0
MatrizPontos[Pallet_2,Prdt_16CoffeCrisp,7].OffsetPlace.C=0
;ENDFOLD
;ENDFOLD

;FOLD PLACE 8
;FOLD PROPRIEDADES
MatrizPontos[Pallet_2,Prdt_16CoffeCrisp,8].NumCaixas = 2
MatrizPontos[Pallet_2,Prdt_16CoffeCrisp,8].PickOp = 1
MatrizPontos[Pallet_2,Prdt_16CoffeCrisp,8].ConfGarraOp = 0
MatrizPontos[Pallet_2,Prdt_16CoffeCrisp,8].FechaGarraOp = 0
MatrizPontos[Pallet_2,Prdt_16CoffeCrisp,8].AbreGarraOp = 0
MatrizPontos[Pallet_2,Prdt_16CoffeCrisp,8].SensoresCaixa = 123
MatrizPontos[Pallet_2,Prdt_16CoffeCrisp,8].TravaGarra = False
MatrizPontos[Pallet_2,Prdt_16CoffeCrisp,8].SkipGoHome = False
MatrizPontos[Pallet_2,Prdt_16CoffeCrisp,8].SkipSobeRelAtual = False
MatrizPontos[Pallet_2,Prdt_16CoffeCrisp,8].XApp1Place=P2_16CoffeCrisp_8_App1
MatrizPontos[Pallet_2,Prdt_16CoffeCrisp,8].XApp2Place=P2_16CoffeCrisp_8_App2
MatrizPontos[Pallet_2,Prdt_16CoffeCrisp,8].XPlace=P2_16CoffeCrisp_8_Place
;ENDFOLD
;FOLD OffsetPlace
MatrizPontos[Pallet_2,Prdt_16CoffeCrisp,8].OffsetPlace.X=0
MatrizPontos[Pallet_2,Prdt_16CoffeCrisp,8].OffsetPlace.Y=0
MatrizPontos[Pallet_2,Prdt_16CoffeCrisp,8].OffsetPlace.Z=0
MatrizPontos[Pallet_2,Prdt_16CoffeCrisp,8].OffsetPlace.A=0
MatrizPontos[Pallet_2,Prdt_16CoffeCrisp,8].OffsetPlace.B=0
MatrizPontos[Pallet_2,Prdt_16CoffeCrisp,8].OffsetPlace.C=0
;ENDFOLD
;ENDFOLD

;ENDFOLD
;ENDFOLD

;FOLD Pallet 2 - Produto 37BarPacking
;FOLD LAYER 1: PLACE 1 ate 2
;FOLD PLACE 1
;FOLD PROPRIEDADES
MatrizPontos[Pallet_2,Prdt_37BarPacking,1].NumCaixas = 3
MatrizPontos[Pallet_2,Prdt_37BarPacking,1].PickOp = 2
MatrizPontos[Pallet_2,Prdt_37BarPacking,1].ConfGarraOp = 2
MatrizPontos[Pallet_2,Prdt_37BarPacking,1].FechaGarraOp = 0
MatrizPontos[Pallet_2,Prdt_37BarPacking,1].AbreGarraOp = 0
MatrizPontos[Pallet_2,Prdt_37BarPacking,1].SensoresCaixa = 123456
MatrizPontos[Pallet_2,Prdt_37BarPacking,1].TravaGarra = False
MatrizPontos[Pallet_2,Prdt_37BarPacking,1].SkipGoHome = False
MatrizPontos[Pallet_2,Prdt_37BarPacking,1].SkipSobeRelAtual = False
MatrizPontos[Pallet_2,Prdt_37BarPacking,1].XApp1Place=P2_37BarPacking_1_App1
MatrizPontos[Pallet_2,Prdt_37BarPacking,1].XApp2Place=P2_37BarPacking_1_App2
MatrizPontos[Pallet_2,Prdt_37BarPacking,1].XPlace=P2_37BarPacking_1_Place
;ENDFOLD
;FOLD OffsetPlace
MatrizPontos[Pallet_2,Prdt_37BarPacking,1].OffsetPlace.X=0
MatrizPontos[Pallet_2,Prdt_37BarPacking,1].OffsetPlace.Y=0
MatrizPontos[Pallet_2,Prdt_37BarPacking,1].OffsetPlace.Z=0
MatrizPontos[Pallet_2,Prdt_37BarPacking,1].OffsetPlace.A=0
MatrizPontos[Pallet_2,Prdt_37BarPacking,1].OffsetPlace.B=0
MatrizPontos[Pallet_2,Prdt_37BarPacking,1].OffsetPlace.C=0
;ENDFOLD
;ENDFOLD

;FOLD PLACE 2
;FOLD PROPRIEDADES
MatrizPontos[Pallet_2,Prdt_37BarPacking,2].NumCaixas = 3
MatrizPontos[Pallet_2,Prdt_37BarPacking,2].PickOp = 2
MatrizPontos[Pallet_2,Prdt_37BarPacking,2].ConfGarraOp = 2
MatrizPontos[Pallet_2,Prdt_37BarPacking,2].FechaGarraOp = 0
MatrizPontos[Pallet_2,Prdt_37BarPacking,2].AbreGarraOp = 0
MatrizPontos[Pallet_2,Prdt_37BarPacking,2].SensoresCaixa = 123456
MatrizPontos[Pallet_2,Prdt_37BarPacking,2].TravaGarra = False
MatrizPontos[Pallet_2,Prdt_37BarPacking,2].SkipGoHome = False
MatrizPontos[Pallet_2,Prdt_37BarPacking,2].SkipSobeRelAtual = False
MatrizPontos[Pallet_2,Prdt_37BarPacking,2].XApp1Place=P2_37BarPacking_2_App1
MatrizPontos[Pallet_2,Prdt_37BarPacking,2].XApp2Place=P2_37BarPacking_2_App2
MatrizPontos[Pallet_2,Prdt_37BarPacking,2].XPlace=P2_37BarPacking_2_Place
;ENDFOLD
;FOLD OffsetPlace
MatrizPontos[Pallet_2,Prdt_37BarPacking,2].OffsetPlace.X=0
MatrizPontos[Pallet_2,Prdt_37BarPacking,2].OffsetPlace.Y=0
MatrizPontos[Pallet_2,Prdt_37BarPacking,2].OffsetPlace.Z=0
MatrizPontos[Pallet_2,Prdt_37BarPacking,2].OffsetPlace.A=0
MatrizPontos[Pallet_2,Prdt_37BarPacking,2].OffsetPlace.B=0
MatrizPontos[Pallet_2,Prdt_37BarPacking,2].OffsetPlace.C=0
;ENDFOLD
;ENDFOLD

;ENDFOLD
;ENDFOLD

;FOLD Pallet 2 - Produto 36BarPacking
;FOLD LAYER 1: PLACE 1 ate 1
;FOLD PLACE 1
;FOLD PROPRIEDADES
MatrizPontos[Pallet_2,Prdt_36BarPacking,1].NumCaixas = 3
MatrizPontos[Pallet_2,Prdt_36BarPacking,1].PickOp = 2
MatrizPontos[Pallet_2,Prdt_36BarPacking,1].ConfGarraOp = 2
MatrizPontos[Pallet_2,Prdt_36BarPacking,1].FechaGarraOp = 0
MatrizPontos[Pallet_2,Prdt_36BarPacking,1].AbreGarraOp = 0
MatrizPontos[Pallet_2,Prdt_36BarPacking,1].SensoresCaixa = 123456
MatrizPontos[Pallet_2,Prdt_36BarPacking,1].TravaGarra = False
MatrizPontos[Pallet_2,Prdt_36BarPacking,1].SkipGoHome = False
MatrizPontos[Pallet_2,Prdt_36BarPacking,1].SkipSobeRelAtual = False
MatrizPontos[Pallet_2,Prdt_36BarPacking,1].XApp1Place=P2_36BarPacking_1_App1
MatrizPontos[Pallet_2,Prdt_36BarPacking,1].XApp2Place=P2_36BarPacking_1_App2
MatrizPontos[Pallet_2,Prdt_36BarPacking,1].XPlace=P2_36BarPacking_1_Place
;ENDFOLD
;FOLD OffsetPlace
MatrizPontos[Pallet_2,Prdt_36BarPacking,1].OffsetPlace.X=0
MatrizPontos[Pallet_2,Prdt_36BarPacking,1].OffsetPlace.Y=0
MatrizPontos[Pallet_2,Prdt_36BarPacking,1].OffsetPlace.Z=0
MatrizPontos[Pallet_2,Prdt_36BarPacking,1].OffsetPlace.A=0
MatrizPontos[Pallet_2,Prdt_36BarPacking,1].OffsetPlace.B=0
MatrizPontos[Pallet_2,Prdt_36BarPacking,1].OffsetPlace.C=0
;ENDFOLD
;ENDFOLD

;ENDFOLD
;ENDFOLD

;FOLD Pallet 2 - Produto 22KitKat
;FOLD LAYER 1: PLACE 1 ate 4
;FOLD PLACE 1
;FOLD PROPRIEDADES
MatrizPontos[Pallet_2,Prdt_22KitKat,1].NumCaixas = 2
MatrizPontos[Pallet_2,Prdt_22KitKat,1].PickOp = 2
MatrizPontos[Pallet_2,Prdt_22KitKat,1].ConfGarraOp = 2
MatrizPontos[Pallet_2,Prdt_22KitKat,1].FechaGarraOp = 0
MatrizPontos[Pallet_2,Prdt_22KitKat,1].AbreGarraOp = 0
MatrizPontos[Pallet_2,Prdt_22KitKat,1].SensoresCaixa = 123
MatrizPontos[Pallet_2,Prdt_22KitKat,1].TravaGarra = False
MatrizPontos[Pallet_2,Prdt_22KitKat,1].SkipGoHome = False
MatrizPontos[Pallet_2,Prdt_22KitKat,1].SkipSobeRelAtual = False
MatrizPontos[Pallet_2,Prdt_22KitKat,1].XApp1Place=P2_22KitKat_1_App1
MatrizPontos[Pallet_2,Prdt_22KitKat,1].XApp2Place=P2_22KitKat_1_App2
MatrizPontos[Pallet_2,Prdt_22KitKat,1].XPlace=P2_22KitKat_1_Place
;ENDFOLD
;FOLD OffsetPlace
MatrizPontos[Pallet_2,Prdt_22KitKat,1].OffsetPlace.X=0
MatrizPontos[Pallet_2,Prdt_22KitKat,1].OffsetPlace.Y=0
MatrizPontos[Pallet_2,Prdt_22KitKat,1].OffsetPlace.Z=0
MatrizPontos[Pallet_2,Prdt_22KitKat,1].OffsetPlace.A=0
MatrizPontos[Pallet_2,Prdt_22KitKat,1].OffsetPlace.B=0
MatrizPontos[Pallet_2,Prdt_22KitKat,1].OffsetPlace.C=0
;ENDFOLD
;ENDFOLD

;FOLD PLACE 2
;FOLD PROPRIEDADES
MatrizPontos[Pallet_2,Prdt_22KitKat,2].NumCaixas = 2
MatrizPontos[Pallet_2,Prdt_22KitKat,2].PickOp = 2
MatrizPontos[Pallet_2,Prdt_22KitKat,2].ConfGarraOp = 2
MatrizPontos[Pallet_2,Prdt_22KitKat,2].FechaGarraOp = 0
MatrizPontos[Pallet_2,Prdt_22KitKat,2].AbreGarraOp = 0
MatrizPontos[Pallet_2,Prdt_22KitKat,2].SensoresCaixa = 123
MatrizPontos[Pallet_2,Prdt_22KitKat,2].TravaGarra = False
MatrizPontos[Pallet_2,Prdt_22KitKat,2].SkipGoHome = False
MatrizPontos[Pallet_2,Prdt_22KitKat,2].SkipSobeRelAtual = False
MatrizPontos[Pallet_2,Prdt_22KitKat,2].XApp1Place=P2_22KitKat_2_App1
MatrizPontos[Pallet_2,Prdt_22KitKat,2].XApp2Place=P2_22KitKat_2_App2
MatrizPontos[Pallet_2,Prdt_22KitKat,2].XPlace=P2_22KitKat_2_Place
;ENDFOLD
;FOLD OffsetPlace
MatrizPontos[Pallet_2,Prdt_22KitKat,2].OffsetPlace.X=0
MatrizPontos[Pallet_2,Prdt_22KitKat,2].OffsetPlace.Y=0
MatrizPontos[Pallet_2,Prdt_22KitKat,2].OffsetPlace.Z=0
MatrizPontos[Pallet_2,Prdt_22KitKat,2].OffsetPlace.A=0
MatrizPontos[Pallet_2,Prdt_22KitKat,2].OffsetPlace.B=0
MatrizPontos[Pallet_2,Prdt_22KitKat,2].OffsetPlace.C=0
;ENDFOLD
;ENDFOLD

;FOLD PLACE 3
;FOLD PROPRIEDADES
MatrizPontos[Pallet_2,Prdt_22KitKat,3].NumCaixas = 2
MatrizPontos[Pallet_2,Prdt_22KitKat,3].PickOp = 2
MatrizPontos[Pallet_2,Prdt_22KitKat,3].ConfGarraOp = 2
MatrizPontos[Pallet_2,Prdt_22KitKat,3].FechaGarraOp = 0
MatrizPontos[Pallet_2,Prdt_22KitKat,3].AbreGarraOp = 0
MatrizPontos[Pallet_2,Prdt_22KitKat,3].SensoresCaixa = 123
MatrizPontos[Pallet_2,Prdt_22KitKat,3].TravaGarra = False
MatrizPontos[Pallet_2,Prdt_22KitKat,3].SkipGoHome = False
MatrizPontos[Pallet_2,Prdt_22KitKat,3].SkipSobeRelAtual = False
MatrizPontos[Pallet_2,Prdt_22KitKat,3].XApp1Place=P2_22KitKat_3_App1
MatrizPontos[Pallet_2,Prdt_22KitKat,3].XApp2Place=P2_22KitKat_3_App2
MatrizPontos[Pallet_2,Prdt_22KitKat,3].XPlace=P2_22KitKat_3_Place
;ENDFOLD
;FOLD OffsetPlace
MatrizPontos[Pallet_2,Prdt_22KitKat,3].OffsetPlace.X=0
MatrizPontos[Pallet_2,Prdt_22KitKat,3].OffsetPlace.Y=0
MatrizPontos[Pallet_2,Prdt_22KitKat,3].OffsetPlace.Z=0
MatrizPontos[Pallet_2,Prdt_22KitKat,3].OffsetPlace.A=0
MatrizPontos[Pallet_2,Prdt_22KitKat,3].OffsetPlace.B=0
MatrizPontos[Pallet_2,Prdt_22KitKat,3].OffsetPlace.C=0
;ENDFOLD
;ENDFOLD

;FOLD PLACE 4
;FOLD PROPRIEDADES
MatrizPontos[Pallet_2,Prdt_22KitKat,4].NumCaixas = 4
MatrizPontos[Pallet_2,Prdt_22KitKat,4].PickOp = 2
MatrizPontos[Pallet_2,Prdt_22KitKat,4].ConfGarraOp = 2
MatrizPontos[Pallet_2,Prdt_22KitKat,4].FechaGarraOp = 0
MatrizPontos[Pallet_2,Prdt_22KitKat,4].AbreGarraOp = 0
MatrizPontos[Pallet_2,Prdt_22KitKat,4].SensoresCaixa = 123456
MatrizPontos[Pallet_2,Prdt_22KitKat,4].TravaGarra = False
MatrizPontos[Pallet_2,Prdt_22KitKat,4].SkipGoHome = False
MatrizPontos[Pallet_2,Prdt_22KitKat,4].SkipSobeRelAtual = False
MatrizPontos[Pallet_2,Prdt_22KitKat,4].XApp1Place=P2_22KitKat_4_App1
MatrizPontos[Pallet_2,Prdt_22KitKat,4].XApp2Place=P2_22KitKat_4_App2
MatrizPontos[Pallet_2,Prdt_22KitKat,4].XPlace=P2_22KitKat_4_Place
;ENDFOLD
;FOLD OffsetPlace
MatrizPontos[Pallet_2,Prdt_22KitKat,4].OffsetPlace.X=0
MatrizPontos[Pallet_2,Prdt_22KitKat,4].OffsetPlace.Y=0
MatrizPontos[Pallet_2,Prdt_22KitKat,4].OffsetPlace.Z=0
MatrizPontos[Pallet_2,Prdt_22KitKat,4].OffsetPlace.A=0
MatrizPontos[Pallet_2,Prdt_22KitKat,4].OffsetPlace.B=0
MatrizPontos[Pallet_2,Prdt_22KitKat,4].OffsetPlace.C=0
;ENDFOLD
;ENDFOLD

